	(*-----------------------Weiterschaltbedingungen----------------------------*)
	IF  NOT fb_xml_srv_read.bBusy  THEN
		IF NOT fb_xml_srv_read.bError THEN
			fb_state_entry.i16_next_step := 30;
		ELSE	(* Fehler *)
			s_PLC_Path_name:='!!! not found !!!';
			nErrId := fb_xml_srv_read.nErrId;
			fb_state_entry.i16_next_step := BEREIT;
			Error_:= TRUE;
		END_IF
	END_IF

	(*PLC Name und Pfad trennen *)
	s_PLC_name:=s_PLC_path_name;
	s_PLC_name:=s_PLC_path_name;
	len_str:=LEN(s_PLC_path_name);
	i:=0;

	FOR i:=1 TO len_str DO
		s_PLC_name:=DELETE(s_PLC_name,FIND(s_PLC_name,'\'),1);
	END_FOR

	s_PLC_path:=s_PLC_path_name;
	s_PLC_path:=DELETE(s_PLC_Path,LEN(s_PLC_path)-FIND(s_PLC_path,s_PLC_name)+1,FIND(s_PLC_path,s_PLC_name));
	s_Projekt_path:=s_PLC_path;

	len_str:=LEN(s_Projekt_path);
	s_Projekt_path:=LEFT(s_Projekt_path, len_str-1);

	(*PLC-Pfad löschen*)
	mid_str:='';
	len_str:=LEN(s_Projekt_path);
	FOR i:=1 TO LEN(s_Projekt_path) DO
			IF		mid_str <> '\' THEN
					s_Projekt_path:=LEFT(s_Projekt_path, len_str-i);
					mid_str:=MID(s_Projekt_path, 1 , len_str-i);
			END_IF
	END_FOR
(*=======================================================*)
30:  fb_state_entry.s_debugtext:='Pfade zusammen bauen';

	IF	s_Projekt_path <> '' THEN
		fb_state_entry.i16_next_step := BEREIT;
	END_IF

	IF	fb_state_entry.X THEN
		IF	FIND(s_tools_path,':') = 0 THEN
			s_tools_path:=CONCAT(s_Projekt_path,s_tools_path);
		END_IF

		IF	FIND(s_ud_path,':') = 0 THEN
			s_ud_path:=CONCAT(s_Projekt_path,s_ud_path);
		END_IF

		IF	FIND(MP_TDPathLocal,':') = 0 THEN
			MP_TDPathLocal:=CONCAT(s_Projekt_path,MP_TDPathLocal);
		END_IF

		IF	FIND(MP_TDPathService,':') = 0 THEN
			MP_TDPathService:=CONCAT(s_Projekt_path,MP_TDPathService);
		END_IF

		IF	FIND(MP_LocalDriveRoot,':') = 0 THEN
			MP_LocalDriveRoot:=CONCAT(s_Projekt_path,MP_LocalDriveRoot);
		END_IF

		IF	FIND(MP_ExportDrive,':') = 0 THEN
			MP_ExportDrive:=LEFT(s_PLC_path_name, 2);
		END_IF

		IF	FIND(MP_ExportDrivePathTD,'_') = 0 THEN
			MP_ExportDrivePathTD:=CONCAT(s_Projekt_path,MP_ExportDrivePathTD);
		END_IF

		IF	FIND(MP_ExportDrivePathMP,'_') = 0 THEN
			MP_ExportDrivePathMP:=CONCAT(s_Projekt_path,MP_ExportDrivePathMP);
		END_IF

		IF	FIND(LOG_RDPathLocal,':') = 0 THEN
			LOG_RDPathLocal:=CONCAT(s_Projekt_path,LOG_RDPathLocal);
		END_IF

		IF	FIND(LOG_ExportDrivePathRD,'_') = 0 THEN
			LOG_ExportDrivePathRD:=CONCAT(s_Projekt_path,LOG_ExportDrivePathRD);
		END_IF

	END_IF

(*=======================================================*)
BEREIT:  fb_state_entry.s_debugtext:='Warten auf Start';

	IF	fb_state_entry.E THEN
		Start:= FALSE;
		Done := TRUE;
	END_IF

	IF	Start THEN
		fb_state_entry.i16_next_step:=INIT;
	END_IF

	IF	fb_state_entry.X THEN
		Done := FALSE;
		Error_:= FALSE;
	END_IF

END_CASE

fb_state_entry(i16_pos:= 2);
(*========================================================================================*)

(* XML *)
fb_xml_srv_read(
	sNetId:= '',
	ePath:= PATH_GENERIC,
	nMode:= XMLSRV_SKIPMISSING,
	sSymName:= ,
	sFilePath:= ,
	sXPath:= ,
	bExecute:= ,
	tTimeout:= t#10s,
	bBusy=> ,
	bError=> ,
	nErrId=> );
END_PROGRAM

(* POU zLibrary/ept/min_exit/ST_MinExit, ST *)
PROGRAM ST_MinExit
VAR
	btn_min					: sButtonVisu;
	btn_exit					: sButtonVisu;

	fb_f_trig_minimieren		: F_TRIG;
	fb_tof_minimieren			: TOF;
	NT_StartProcess 			: NT_StartProcess;
	s_comndline						:STRING(255);
END_VAR
(*
in der C:\TwinCAT\Plc\TwinCAT PLC Control.ini muss
NoFullScreenMode=No umgestellt werden
=====================================================================*)



btn_min.Text:='_';
btn_min.Enable:=FALSE;
IF	btn_min.Pressed THEN
	btn_min.BackgroundColor:=Color.darkgrey;
ELSE
	btn_min.BackgroundColor:=Color.lightgrey;
END_IF
btn_min.TextColor:=Color.black;
btn_min.Visible:=FALSE;
fb_f_trig_minimieren(CLK:=btn_min.Pressed);
fb_tof_minimieren(IN:=fb_f_trig_minimieren.Q,PT:=t#1s);

IF	fb_f_trig_minimieren.Q THEN
	NT_StartProcess.START:=TRUE;
END_IF
IF 	NT_StartProcess.BUSY THEN
	NT_StartProcess.START:=FALSE;
END_IF

		(*minimieren wird mit vbs Skript gestartet*)
	NT_StartProcess(
			NETID:=,
			PATHSTR	:='C:\Windows\System32\wscript.exe',
			DIRNAME	:=s_tools_path,
			COMNDLINE	:='minimieren.vbs',
			START		:=,
			TMOUT		:=T#10s);
(*=====================================================================*)
btn_exit.Text:='X';
btn_exit.Enable:=FALSE;
IF	btn_exit.Pressed THEN
	btn_exit.BackgroundColor:=Color.darkgrey;
ELSE
	btn_exit.BackgroundColor:=Color.lightgrey;
END_IF

btn_exit.TextColor:=Color.black;
btn_exit.Visible:=FALSE;
END_PROGRAM

(* POU zLibrary/ept/ST_SaveAndLoad, ST *)
PROGRAM ST_SaveAndLoad
VAR_OUTPUT
	st_ctrl_out			:struct_ctrl_out;
END_VAR
VAR
	b_init				:BOOL;
	fb_state_entry		:ST_StateEntry;
	fb_ton_quitt		:TON;

	NT_StartProcess 	:NT_StartProcess;
	fbFileDelete		:FB_FileDelete;

	s_script			:STRING;

	btn_load			:sButtonVisu;
	btn_save			:sButtonVisu;

END_VAR
VAR CONSTANT
		s_bbgenMachineToSrv				:STRING:=		'_TD_save.bat';
		s_bbgenSrvToMachine				:STRING:=		'_TD_load.bat';

END_VAR
(*======================================================
   ST_SaveAndLoad
 ------------------------------------------------------
   Auth: 		Werner Friedl   						 
   Date: 		06.10.2020   						     
   Rev.: 		1.0	
   Desc:		Die bat Datein zum laden und speichern der BBgen Dateien werden hier ausgeführt.
			mit der Constante b_wkzBereinigen kann bestimmt werden, ob die Werkzeugdateu vorher gelöscht wird.

 ========================================================*)
IF	NOT b_init THEN
	b_Init:=TRUE;
END_IF
CallPrg();
Btn_init();
(* ========================================================*)
fb_ton_quitt(IN:= , PT:= t#100ms, Q=> , ET=> );

fb_state_entry(i16_pos:= 1);
CASE fb_state_entry.i16_step OF
(*=======================================================*)
INIT_OBJ:
		fb_state_entry.i16_next_step := INIT;

(*=======================================================*)
INIT:
	fb_state_entry.i16_next_step := BEREIT;

(*=======================================================*)
BEREIT:	fb_state_entry.s_debugtext:='warte auf Taster Save oder Load';

	IF fb_state_entry.E THEN
		st_ctrl_out.b_bereit:=TRUE;
		NT_StartProcess.START:=FALSE;
	END_IF

	(*-----------------------Weiterschaltbedingungen----------------------------*)
	IF 	btn_load.Pressed THEN
		fb_state_entry.i16_next_step:=110;
		s_script:=CONCAT(CURRENTLANGUAGE,s_bbgenSrvToMachine);
	ELSIF
		btn_save.Pressed THEN
		s_script:=CONCAT(CURRENTLANGUAGE,s_bbgenMachineToSrv);
		fb_state_entry.i16_next_step:=110;
	END_IF


	IF fb_state_entry.X THEN
		st_ctrl_out.b_busy:=TRUE;
		st_ctrl_out.b_bereit := FALSE;
		st_ctrl_out.b_fertig := FALSE;
	END_IF

(*=======================================================*)
110:fb_state_entry.s_debugtext:='start bat Script "Laden der Dateien vom Server"';

	IF 	fb_state_entry.E THEN
		NT_StartProcess.START:=TRUE;
	END_IF

	(*-----------------------Weiterschaltbedingungen----------------------------*)
	IF 	NT_StartProcess.BUSY THEN
		fb_state_entry.i16_next_step:=120;
	END_IF

	IF 	fb_state_entry.X THEN
		NT_StartProcess.START:=FALSE;
	END_IF

(*=======================================================*)
120:fb_state_entry.s_debugtext:='Warten auf fertig';

	IF	NOT btn_load.Pressed AND
		NOT btn_save.Pressed  THEN
		IF 	NT_StartProcess.ERR THEN
			fb_state_entry.s_debugtext:=CONCAT(fb_state_entry.s_debugtext,' ERRID => ');
			fb_state_entry.s_debugtext:=CONCAT(fb_state_entry.s_debugtext,UDINT_TO_STRING(NT_StartProcess.ERRID));
			fb_state_entry.i16_next_step:=FEHLER;
		ELSIF
			NOT NT_StartProcess.BUSY AND
			NOT NT_StartProcess.ERR AND
			fb_state_entry.fb_ton_Step.ET>t#3000ms THEN
			st_ctrl_out.b_busy:=FALSE;
			st_ctrl_out.b_fertig := TRUE;
			fb_state_entry.i16_next_step:=BEREIT;
		END_IF
	END_IF

(*=======================================================*)
STOP, FEHLER:

	IF fb_state_entry.E THEN
		st_ctrl_out.b_fehler := fb_state_entry.i16_step = FEHLER;
		st_ctrl_out.b_gestoppt := fb_state_entry.i16_step = STOP;
		st_ctrl_out.b_busy:=FALSE;
	END_IF

	IF	fb_state_entry.fb_ton_Step.ET > t#1000ms THEN   (*Quittiert sich selbst*)
		fb_state_entry.i16_next_step:=INIT;
	END_IF

END_CASE

fb_state_entry(i16_pos:= 2 );
END_PROGRAM
ACTION Btn_init:
btn_load.Text:='loadSrv';
btn_load.Enable:=CurrentUserLevel >=6 AND ModeSelect.Mode<=MODE_MANUAL;
IF btn_load.Enable THEN
	btn_load.TextColor:=Color.black;
ELSE
	btn_load.TextColor:=Color.grey;
END_IF
btn_load.Visible:= TRUE;

IF	btn_load.Pressed THEN
	btn_load.BackgroundColor:=Color.grey;
ELSE
	btn_load.BackgroundColor:=Color.lightgrey;
END_IF



btn_save.Text:='saveSrv';
btn_save.Enable:=CurrentUserLevel >=6 AND ModeSelect.Mode<=MODE_MANUAL;
IF btn_save.Enable THEN
	btn_save.TextColor:=Color.black;
ELSE
	btn_save.TextColor:=Color.grey;
END_IF
btn_save.Visible:= TRUE;

IF	btn_save.Pressed THEN
	btn_save.BackgroundColor:=Color.grey;
ELSE
	btn_save.BackgroundColor:=Color.lightgrey;
END_IF
END_ACTION
ACTION CallPrg:
NT_StartProcess(
	NETID:='',
	PATHSTR		:='C:\Windows\System32\cmd.exe',
	DIRNAME		:=s_tools_path,
	COMNDLINE	:=CONCAT('/C start /b ', s_script),
	START			:=,
	TMOUT			:=DEFAULT_ADS_TIMEOUT);


fbFileDelete(
	sNetId:= ,
	sPathName:= , 
	ePath:= PATH_GENERIC,
	bExecute:= ,
	tTimeout:= t#1s );
END_ACTION

(* POU zLibrary/ept/BDE/ST_Hydra8, ST *)
PROGRAM ST_Hydra8
VAR
	fb_tof_produktion			: TOF;
	fb_r_trig_signal			: R_TRIG;

	a_signal_produktion				AT %Q* : BOOL;
	a_signal_gutteil				AT %Q* : BOOL;
	a_signal_schlechtteil			AT %Q* : BOOL;
	a_signal_reserve				AT %Q* : BOOL;
	a_Fehlerfeld					: DWORD := 0;
END_VAR
(* Zeiten *)
fb_tof_produktion(
				IN:= 	(fb_r_trig_signal.Q AND
				ModeSelect.Mode=MODE_AUTO_RUN) OR
				(ST02_S1_40K01.BitInToCheck),
				PT:= T#60s,
				Q=>  a_signal_produktion,
				ET=> );

(* Flanken *)
IF	ST_CPU.LNG =CZ THEN
	fb_r_trig_signal(	CLK:= Robot01.State = STATE_OK);
END_IF

st_Hydra8Data.bStatus[_PRODUKTION] := a_signal_produktion;
END_PROGRAM

(* POU zLibrary/ept/BDE/ST_ImportHydraString, ST *)
PROGRAM ST_ImportHydraString
VAR_INPUT
	s_Path				: T_MaxString;
	sDateiName			: STRING;
	tStartTime			: TIME := T#10S;
END_VAR
VAR
	fb_state_entry			: ST_StateEntry;
	fbFindFiles			: FB_EnumFindFileList;
	fbFindFilesEntry		: ST_FindFileEntry;
	fbFileOpen			: FB_FileOpen;
	fbFileGets			: FB_FileGets;
	fbFileClose			: FB_FileClose;
	fbFileDelete			: FB_FileDelete;
	HelpString			: T_MaxString;
	fb_ton_start			: TON;
	hFile				:UINT:=0;
	nErrIdOpen			:UDINT;
	nErrIdRead			:UDINT;
	nErrIdClose			:UDINT;
	nErrIdDelete			:UDINT;
	sFileName			:STRING;

	iHelp				: INT;

	(* Für Anzeige in Visu *)
	iProduktionssperre	: INT;	(* 0 = nicht aktiv, 1 = aktiv, 2 = Status ungültig *)
END_VAR
VAR_OUTPUT
	Ready						:BOOL;
	Busy						:BOOL;
	Done						:BOOL;
	Error						:BOOL;
END_VAR
VAR CONSTANT
	sDatumPrefix				: STRING := 'DAT=';
	sZeitPrefix				: STRING := 'ZEI=';
	sOutput					: STRING := 'OUT';
	sTrennzeichen			: STRING := '|';
END_VAR
(*======================================================
   ST: ST_Import_Hydra_String
 ------------------------------------------------------
   Auth: 	Thomas Vilgis    						 
   Date: 	02.02.2022    						     
   Rev.: 	1.0	
   Desc:		Es wird alle 10 Sekunden (Zeit im Aufruf einstellbar) eine Textdatei mit 8 Status Ausgänge von Hydra erstellt.
			TwinCAT liest diese Datei aus und löscht sie dann.
			Es gibt nur eine Zeile in der Textdatei.
			Der erste Ausgang ist für den Status der Produktionssperre.
			Ein OUT Status steht nur in der Datei, wenn es eine Änderung gegeben hat.	
				
			So sieht die Datei aus: (alles in einer Zeile)
			OUT1=0|OUT2=0|OUT3=0|OUT4=0|OUT5=0|
			OUT6=0|OUT7=0|OUT8=0|DAT=02.02.2021|ZEI=07:16:00

   Historie: 	1.0

 ========================================================*)



(* Zeiten *)
fb_ton_start(IN:= NOT fb_ton_start.Q, PT:= tStartTime, Q=>  , ET=> );


(* ======================================Schrittkette======================================== *)
fb_state_entry(i16_pos:= 1);

CASE fb_state_entry.i16_step OF
(*=======================================================*)
	INIT_OBJ: fb_state_entry.s_debugtext:='initialisieren';

		(*-----------------------Weiterschaltbedingungen----------------------------*)
		IF fb_state_entry.fb_ton_Step.ET >= T#5S THEN
			fb_state_entry.i16_next_step:=BEREIT;
		END_IF

(*=======================================================*)
	BEREIT: fb_state_entry.s_debugtext:='Start';

		IF fb_state_entry.E THEN
			Ready := TRUE;
		END_IF

		(*-----------------------Weiterschaltbedingungen----------------------------*)
		IF fb_ton_start.Q THEN
			Error := FALSE;
			Busy := TRUE;
			Ready := FALSE;
			Done := FALSE;
			fb_state_entry.i16_next_step:=110;
		END_IF
		
		IF fb_state_entry.X THEN
			sFileName:=CONCAT(s_Path,sDateiName);
		END_IF
		
(*=======================================================*)
	110: fb_state_entry.s_debugtext:='HelpString löschen';
	
		IF fb_state_entry.E THEN
			HelpString := '';
		END_IF

		(*-----------------------Weiterschaltbedingungen----------------------------*)
		fb_state_entry.i16_next_step:=120;

(*=======================================================*)
	120: fb_state_entry.s_debugtext:='Prüfe, ob Datei vorhanden ist';

		IF fb_state_entry.E THEN
			fbFindFiles.bExecute := TRUE;
		END_IF

		(*-----------------------Weiterschaltbedingungen----------------------------*)
		IF fbFindFiles.bBusy THEN
			fb_state_entry.i16_next_step:=130;
		END_IF

(*=======================================================*)
	130: fb_state_entry.s_debugtext:='Prüfe, ob Datei vorhanden ist';

		(*-----------------------Weiterschaltbedingungen----------------------------*)
		IF NOT fbFindFiles.bBusy THEN
			fbFindFiles.bExecute := FALSE;
			IF NOT fbFindFiles.bError THEN
				IF fbFindFiles.nFindFiles = 1 THEN
					fb_state_entry.i16_next_step:=140;
				ELSE
					fb_state_entry.i16_next_step:=240;	(* Datei nicht vorhanden >> Auswertung *)
				END_IF
			ELSE
				fb_state_entry.i16_next_step:=FEHLER;
			END_IF
		END_IF

(*=======================================================*)
	140: fb_state_entry.s_debugtext:='Datei öffnen';

		IF fb_state_entry.E THEN
		   	fbFileOpen.bExecute:=TRUE;
		END_IF

		(*-----------------------Weiterschaltbedingungen----------------------------*)
		IF fbFileOpen.bBusy THEN
			fb_state_entry.i16_next_step:=150;
		END_IF

(*=======================================================*)
	150: fb_state_entry.s_debugtext:='Datei öffnen';

		(*-----------------------Weiterschaltbedingungen----------------------------*)
		IF 	NOT fbFileOpen.bBusy THEN

			fbFileOpen.bExecute:=FALSE;
			IF 	fbFileOpen.bError THEN
				nErrIdOpen:=fbFileOpen.nErrId;
				fb_state_entry.i16_next_step:=200;
			ELSE
				hFile := fbFileOpen.hFile;	(* Sehr wichtig hFile für FileRead und Fileclose übergeben *)
				fb_state_entry.i16_next_step:=160;
			END_IF
		END_IF

(*=======================================================*)
	160: fb_state_entry.s_debugtext:='Datei auslesen';

		IF fb_state_entry.E THEN
			fbFileGets.bExecute:=TRUE;
		END_IF

		(*-----------------------Weiterschaltbedingungen----------------------------*)
		IF  fbFileGets.bBusy THEN
			fb_state_entry.i16_next_step:=170;
		END_IF

(*=======================================================*)
	170: fb_state_entry.s_debugtext:='Datei auslesen';

		(*-----------------------Weiterschaltbedingungen----------------------------*)
		IF 	NOT fbFileGets.bBusy THEN
			fbFileGets.bExecute:=FALSE;
			IF 	fbFileGets.bError THEN
				nErrIdRead:=fbFileGets.nErrId;
				fb_state_entry.i16_next_step:=200;
			ELSE
				HelpString := fbFileGets.sLine;
				fb_state_entry.i16_next_step:=200;
			END_IF
		END_IF

(*=======================================================*)
	200: fb_state_entry.s_debugtext:='Datei schließen';

		IF fb_state_entry.E THEN
			fbFileClose.bExecute:=TRUE;
		END_IF

		(*-----------------------Weiterschaltbedingungen----------------------------*)
		IF 	fbFileClose.bBusy THEN
			fb_state_entry.i16_next_step:=210;
		END_IF

(*=======================================================*)
	210: fb_state_entry.s_debugtext:='Datei schließen';

		(*-----------------------Weiterschaltbedingungen----------------------------*)
		IF NOT fbFileClose.bBusy THEN
			fbFileClose.bExecute:=FALSE;
			IF 	fbFileClose.bError THEN
				nErrIdClose:=fbFileClose.nErrId;
				fb_state_entry.i16_next_step:=FEHLER;
			ELSE
				hFile := 0;
				fb_state_entry.i16_next_step:=220;
			END_IF
		END_IF
		
(*=======================================================*)
	220: fb_state_entry.s_debugtext:='Datei löschen';

		IF fb_state_entry.E THEN
			fbFileDelete.bExecute:=TRUE;
		END_IF

		(*-----------------------Weiterschaltbedingungen----------------------------*)
		IF 	fbFileDelete.bBusy THEN
			fb_state_entry.i16_next_step:=230;
		END_IF

(*=======================================================*)
	230: fb_state_entry.s_debugtext:='Datei löschen';

		(*-----------------------Weiterschaltbedingungen----------------------------*)
		IF NOT fbFileDelete.bBusy THEN
			fbFileDelete.bExecute:=FALSE;
			IF 	fbFileDelete.bError THEN
				nErrIdDelete:=fbFileDelete.nErrId;
				fb_state_entry.i16_next_step:=FEHLER;
			ELSE
				fb_state_entry.i16_next_step:=240;
			END_IF
		END_IF

(* Falls die Auswertung der Datei für jede Anlage unterschiedlich ist,
sollte man die Auswertung in einem eigenen Baustein machen *)
(*=======================================================*)
	240: fb_state_entry.s_debugtext:='Auswertung, ob Produktionssperre aktiv ist';

		IF fb_state_entry.E THEN
			IF fbFindFiles.nFindFiles = 0 THEN	(* Datei war gar nicht vorhanden *)
				iProduktionssperre := 2;	(* Status ungültig *)
			ELSE
				(* Suche nach OUT1= *)
				iHelp := FIND(HelpString, CONCAT(sOutput, '1='));
				IF iHelp > 0 THEN
					IF MID(HelpString, 1, 6) = '0' THEN	(* an Stelle 6 steht 0 oder 1 *)
						iProduktionssperre := 0;	(* nicht aktiv *)
					ELSIF MID(HelpString, 1, 6) = '1' THEN	(* an Stelle 6 steht 0 oder 1 *)
						iProduktionssperre := 1;	(* aktiv *)
					END_IF
				END_IF
			END_IF
		END_IF

		(*-----------------------Weiterschaltbedingungen----------------------------*)
		Busy := FALSE;
		Done := TRUE;
		fb_state_entry.i16_next_step:=BEREIT;
		
	

(*=======================================================*)
	FEHLER:
		IF fb_state_entry.E THEN
			Error := TRUE;
		END_IF

		(*-----------------------Weiterschaltbedingungen----------------------------*)
		fb_state_entry.i16_next_step:=BEREIT;

END_CASE


fb_state_entry(i16_pos:= 2);


fbFindFiles(
	bExecute	:= ,
	sNetId		:= '',
	sPathName	:= sFileName,
	pFindList	:= ADR(fbFindFilesEntry),
	cbFindList	:= SIZEOF(fbFindFilesEntry),
	tTimeout	:= t#1s );

 fbFileOpen(
	sNetId:='',
	sPathName:= sFileName,
	nMode:=FOPEN_MODEREAD,
	ePath:=PATH_GENERIC,
	bExecute:= ,
	tTimeout:=T#1s,
	hFile=> );

fbFileGets(
	sNetId:= , 
	hFile:= hFile, 
	bExecute:= , 
	tTimeout:= , 
	bBusy=> , 
	bError=> , 
	nErrId=> , 
	sLine=> , 
	bEOF=> );

fbFileClose(
	sNetId:='',
	hFile:=hFile,
	bExecute:= ,
	tTimeout:=T#1S);
	
fbFileDelete(
	sNetId:= , 
	sPathName:= sFileName, 
	ePath:= PATH_GENERIC, 
	bExecute:= , 
	tTimeout:= , 
	bBusy=> , 
	bError=> , 
	nErrId=> );
END_PROGRAM

(* POU System/LoginDialog/ImpExp_UD, ST *)
PROGRAM ImpExp_UD
VAR_INPUT
	Start_write				:BOOL;
	Start_read				:BOOL;
	path					:STRING(255);
	filename					:STRING(255);
END_VAR
VAR
	b_init					:BOOL;
	fb_state_entry				:ST_StateEntry;

	fb_xml_srv_read			: FB_XmlSrvReadByName;
	fb_xml_srv_write			: FB_XmlSrvWriteByName;

	fb_rtrig_Start_read			:R_TRIG;
	fb_rtrig_Start_write_to_server:R_TRIG;
	fb_ton_init				:TON;
	fb_ton_wz				:TON;
	fb_ton_uez				:TON;

	bError					: BOOL;
	nErrId					: UDINT;
	s_info					: STRING;
	MsgOK					: BOOL;
	MsgID					:STRING(20);

	UserList_Copy			: ARRAY [1..NO_OF_USERS] OF sUserData;

END_VAR

VAR_OUTPUT
	Busy					:BOOL;
	Done					:BOOL;
	Error					:BOOL;
	ErrorMsg				:STRING(255);
END_VAR

VAR CONSTANT
	SymName				:STRING:='.UD';
	xPath					:STRING:='/UD';
END_VAR

VAR_IN_OUT

END_VAR
(*======================================================
   PRG: XML Import und Export der UD
 ------------------------------------------------------
   Auth: 		Werner Friedl    						 
   Date: 		05.01.2021  						     
   Rev.: 		1.0	
   Desc:		
	- Userdate werden beim Neustart eingelesen
	- bei einer Änderung wird Änderung automatisch in die xml eingeragen

   Historie:   1.0

 ========================================================*)
fb_ton_init(IN:= TRUE, PT:=t#1500ms , Q=> , ET=> );
IF	NOT b_init AND fb_ton_init.Q THEN
	Start_read := TRUE;
	b_Init:=TRUE;
END_IF

(* ========================================================*)
fb_rtrig_Start_read();
IF	fb_rtrig_Start_read.Q AND
	NOT Start_write THEN
	Start_read:=TRUE;
END_IF

IF 	(MEMCMP(ADR(UserList_Copy),ADR(UD.UserList),SIZEOF(UserList_Copy))<>0)AND (*automatisch speichern im Manualmode*)
     	ModeSelect.Mode <=MODE_MANUAL AND
	NOT Start_read AND
	b_Init THEN
	Start_write := TRUE;
END_IF

(* ========================================================*)
fb_ton_wz(IN:= , PT:=t#3000ms , Q=> , ET=> );
IF	fb_ton_wz.Q THEN
	fb_ton_wz.IN:=FALSE;
	s_info := '';
END_IF

fb_state_entry(i16_pos:= 1);
CASE fb_state_entry.i16_step OF

(*=======================================================*)
0:	(*initialisieren*)
	Start_write := FALSE;
	Start_read := FALSE;
	fb_state_entry.i16_next_step:=BEREIT;

(*=======================================================*)
BEREIT: fb_state_entry.s_debugtext:='warte auf start';

	IF	Start_read THEN
		fb_state_entry.i16_next_step:=110;
	END_IF

	IF	Start_write THEN
		fb_state_entry.i16_next_step:=200;
	END_IF

	IF fb_state_entry.X THEN
		fb_ton_uez.IN:=FALSE;
		Start_write:=FALSE;
		Start_read:=FALSE;
		Busy:=TRUE;
		Error:=FALSE;
		Done:=FALSE;
		nErrId:=0;
		ErrorMsg:='';
		MsgID:='';
	END_IF

(*=======================================================*)
110: fb_state_entry.s_debugtext:='XML auslesen';	 

	IF fb_state_entry.E THEN
		fb_xml_srv_read.sFilePath := CONCAT(path,filename);
		fb_xml_srv_read.sSymName:=SymName;
		fb_xml_srv_read.sXPath :=xPath;
		fb_xml_srv_read.bExecute := TRUE;
	END_IF

	IF fb_xml_srv_read.bBusy THEN
		fb_xml_srv_read.bExecute := FALSE;
		fb_state_entry.i16_next_step := 120;
	END_IF

(*=======================================================*)
120: fb_state_entry.s_debugtext:='Lesevorgang erfolgreich?';

	IF  NOT fb_xml_srv_read.bBusy  THEN
		IF NOT fb_xml_srv_read.bError THEN
			fb_state_entry.i16_next_step := 900;
		ELSE	(* Fehler *)
			nErrId := fb_xml_srv_read.nErrId;
			IF	nErrId =1804 THEN
				MsgID:='PM15';
				ErrorMsg:='Die Datei UD.xml ist nicht vorhanden';
				fb_state_entry.i16_next_step := 200;	(*Datei wird erstellt*)
			ELSE
				MsgID:='PM16';
				ErrorMsg:='Fehler beim Einlesen der UD.xml Datei';
				fb_state_entry.i16_next_step := FEHLER;
			END_IF
		END_IF
	END_IF

	IF fb_state_entry.X THEN
		fb_ton_wz.IN:=TRUE;
		s_info:=CONCAT('read ',filename);
	END_IF

(*=======================================================*)
200: fb_state_entry.s_debugtext:='XML schreiben';

	IF fb_state_entry.E THEN
		fb_xml_srv_write.sFilePath := CONCAT(path,filename);
		fb_xml_srv_write.sSymName:=SymName;
		fb_xml_srv_write.sXPath :=xPath;
		fb_xml_srv_write.bExecute := TRUE;
	END_IF

	IF fb_xml_srv_write.bBusy THEN
		fb_xml_srv_write.bExecute := FALSE;
		fb_state_entry.i16_next_step := 220;
	END_IF

(*=======================================================*)
220: fb_state_entry.s_debugtext:='Schreiben erfolgreich?';

	IF  NOT fb_xml_srv_write.bBusy  THEN
		IF NOT fb_xml_srv_write.bError THEN
			UserList_Copy := UD.UserList;
			fb_state_entry.i16_next_step := 900;
		ELSE	(* Fehler *)
			nErrId := fb_xml_srv_write.nErrId;
			MsgID:='PM17';
			ErrorMsg:='Fehler beim Schreiben der UD.xml';
			fb_state_entry.i16_next_step := FEHLER;
		END_IF
	END_IF

	IF fb_state_entry.X THEN
		fb_ton_wz.IN:=TRUE;
		fb_ton_uez.IN:=TRUE;		(*automatisch auf Server speichern*)
		s_info:=CONCAT('write ',filename);
	END_IF

(*=======================================================*)
900: fb_state_entry.s_debugtext:='Fertig';

	Busy:=FALSE;
	Done:=TRUE;
	fb_state_entry.i16_next_step:=0;

(*=======================================================*)
FEHLER:

	IF fb_state_entry.E THEN
		MessageHandler.ClearMessageLines(sVisu:=Visu.Message);
	END_IF
	MessageHandler.Msg.ID:=MsgID;
	MessageHandler.Msg.Name:=ErrorMsg;
	MessageHandler.Msg.Text:=ErrorMsg;
	MessageHandler.Msg.Color:=Color.red;
	MessageHandler.Msg.Station:=0;

	MessageHandler(
		Prio:=2, 							(*1=highest, .. , 4=lowest*)
		Btn1Addr:=ADR(MsgOk),			(*Address of Button1 , if Zero then Button is unvisible*)
		Btn2Addr:=,						(*Address of Button2 , if Zero then Button is unvisible*)
		sVisu:=Visu.Message);

	IF MsgOK THEN
		MsgOk:=FALSE;
		fb_state_entry.i16_next_step:=0;
		Busy:=FALSE;
		Error:=TRUE;
	END_IF
END_CASE

fb_state_entry(i16_pos:= 2);


fb_xml_srv_read(
	sNetId:= '',
	ePath:= PATH_GENERIC,
	nMode:= XMLSRV_SKIPMISSING,
	sSymName:= ,
	sFilePath:= ,
	sXPath:= ,
	bExecute:= ,
	tTimeout:= t#10s,
	bBusy=> ,
	bError=> ,
	nErrId=> );

fb_xml_srv_write(
	sNetId:= '',
	ePath:= PATH_GENERIC,
	nMode:= XMLSRV_ADDMISSING,
	sSymName:=  ,
	sFilePath:= ,
	sXPath:= ,
	bExecute:= ,
	tTimeout:= t#10s,
	bBusy=> ,
	bError=> ,
	nErrId=> );


(*automatisch auf Server speichern=============================================*)
fb_ton_uez(PT:=t#20s);
fb_rtrig_Start_write_to_server(CLK:=fb_ton_uez.Q , Q=> );
(*
NT_StartProcess(
	NETID:='',
	PATHSTR	:='C:\Windows\System32\cmd.exe',
	DIRNAME	:='D:\Tools ',
	COMNDLINE	:='/C copy C:\MP\MachPara.xml \\10.16.50.9\bbgen\UML3\MD & @ping localhost -n 4 >NUL',
	START		:=fb_rtrig_Start_write_to_server.Q,
	TMOUT		:=t#10s);
*)
(*
NT_StartProcess(
	NETID:='',
	PATHSTR	:='C:\Windows\System32\wscript.exe',
	DIRNAME	:='D:\Tools',
	COMNDLINE	:='de_PD_aktuell_von_uml_nach_server.vbs',
	START		:=fb_rtrig_Start_write_to_server.Q,
	TMOUT		:=t#10s);
*)
END_PROGRAM

(* POU System/LoginDialog/UserLoginHandler, ST *)
PROGRAM UserLoginHandler
VAR
	Keypad								: UserLoginKeypad;
	btn_Login							: VisuButton;
	btn_LogOut							: VisuButton;
	btn_ChangeUserData				: VisuButton;
	btn_ChangePassword				: VisuButton;

	PasswordChangeActive				: BOOL;

	UserListIndexFixed					: INT;
	FixUserList							: BOOL;
	FP_FixUserList						: R_TRIG;
	FP_PasswordChangeActive			: R_TRIG;

	SelectedUser						: sUserData;
	UserLoggedOut						: sUserData;
	EmptyUser							: sUserData;

	CurrentVisuOld						: STRING;
	UserListIndexOld					: INT;

	InfoLogin              					: ErrorStruct;
	InfoLogout           					: ErrorStruct;

	TP_LogegdIn						: TP;
	TP_LogegdOut						: TP;

	Index								: INT;

	ton_AutoLoggedOut					: TON;
	b_Button							: BOOL;
	CopyCurrentVisu						: STRING;
	s_AutoLoggedOut					: STRING;

END_VAR
VAR_IN_OUT
	sVisu								: sVisuLoginDialog;
	UserList								: ARRAY [1..NO_OF_USERS] OF sUserData;

END_VAR
VAR_OUTPUT
	CurrentUser							: sUserData;
	UserLoggedIn						: BOOL;
END_VAR
(* Fix Administrator and Operator *)
UserList[1].UserName							:= 'Administrator';
(*UserList[1].UserPassword						:= '123';*)			(*PW in der ".....\UD\UserList.xml  " ändern und PLC neu starten*)
UserList[1].UserLevel							:= 7;
UserList[1].UserCanChangeOwnPassword			:= FALSE;

UserList[2].UserName							:= 'Service';
UserList[2].UserLevel							:= 6;
UserList[2].UserCanChangeOwnPassword			:= FALSE;

(* Fix UserLoggedOut *)
UserLoggedOut.UserName						:= 'Produktion';(*'Logged out';*)
UserLoggedOut.UserPassword					:= '';
UserLoggedOut.UserLevel						:= 1;
UserLoggedOut.UserCanChangeOwnPassword	:= FALSE;



Keypad(sVisu:= sVisu.LoginKeyPad,HidePasswordString:=NOT PasswordChangeActive);

FixUserList:= Keypad.Visible OR
			(CurrentUser.UserName<>UserLoggedOut.UserName AND CurrentUserLevel<6);

FP_FixUserList(CLK:= FixUserList );


(* Save Selecte UserIndex from Visu *)
IF 	FP_FixUserList.Q THEN
	UserListIndexFixed:=sVisu.UserListIndex;
END_IF;

(* Disable Selection in sVisu  *)
IF 	FixUserList THEN
	sVisu.UserListIndex:=UserListIndexFixed;
ELSE
	IF	sVisu.UserListIndex > 0 THEN
		SelectedUser:=UserList[sVisu.UserListIndex];
	END_IF
END_IF


(* Handle Keypad *)
FP_PasswordChangeActive(CLK:= PasswordChangeActive);
IF 	btn_Login.PressedFlag AND SelectedUser.UserPassword<>'' OR	(*Login with PW*)
	FP_PasswordChangeActive.Q THEN								(*PW-Change*)
	Keypad.Visible:=TRUE;
END_IF

IF 	Keypad.btnESC OR Keypad.btnOK OR CurrentVisuOld<>CurrentVisu THEN
	Keypad.Visible:=FALSE;
END_IF


(* Handle Login / Logout *)
btn_Login	(TextOn:= 'Login',	Button:= sVisu.btn_Login );
btn_LogOut	(TextOn:= 'Logout',	Button:= sVisu.btn_LogOut );

btn_Login.Enable:=TRUE;

btn_LogOut.Enable:=CurrentUser.UserName<>UserLoggedOut.UserName AND NOT PasswordChangeActive;


IF btn_LogOut.PressedFlag THEN
	(* Generate information Errorlog *)
	InfoLogout.Text			:=  CONCAT('LoginHandler: User ausgeloggt:',CurrentUser.UserName);
	InfoLogout.Typ			:=  2;
	InfoLogout.No			:=  1;
	InfoLogout.DateTime	:=  gVarDTSystemtime;
	TP_LogegdOut.IN		:= TRUE;

	CurrentUserLevel		:= 0;
	CurrentUser				:= UserLoggedOut;
END_IF

(*LogIn finished ok*)
IF 	Keypad.btnOK AND Keypad.InputString=SelectedUser.UserPassword AND NOT PasswordChangeActive OR		(*Login with PW, and PW ok*)
	btn_Login.PressedFlag AND SelectedUser.UserPassword='' THEN												(*Login without PW*)
	CurrentUserLevel		:= SelectedUser.UserLevel;
	CurrentUser				:= SelectedUser;
	(* Generate information Errorlog *)
	InfoLogin.Text			:= CONCAT('LoginHandler: User eingeloggt:',CurrentUser.UserName);
	InfoLogin.Typ			:= 2;
	InfoLogin.No			:= 1;
	InfoLogin.DateTime		:= gVarDTSystemtime;
	TP_LogegdIn.IN			:= TRUE;
END_IF


(* Edit Userlist *)

(* Show Edit Fields *)
sVisu.ShowEditFields:=(sVisu.UserListIndex>=2 AND CurrentUserLevel=7) OR (sVisu.UserListIndex>=3 AND CurrentUserLevel=6);

btn_ChangeUserData(Button:= sVisu.btn_ChangeUserData );
btn_ChangeUserData.Visible:=sVisu.ShowEditFields;

IF 	sVisu.UserEdit.UserName='' THEN
	btn_ChangeUserData.TextOn:= 'ChangeUserDataDel';
ELSE
	btn_ChangeUserData.TextOn:= 'ChangeUserData';
END_IF

IF 	btn_ChangeUserData.PressedFlag THEN
	(* Take new Userdatas when Username is not Administrator and Produktion *)
	IF 	sVisu.UserEdit.UserName <> 'Administrator' AND sVisu.UserEdit.UserName <> 'Produktion' THEN
		UserList[sVisu.UserListIndex]:=sVisu.UserEdit;
		IF 	UserList[sVisu.UserListIndex].UserName=''  THEN
			FOR index:= sVisu.UserListIndex TO DINT_TO_INT(NO_OF_USERS-1) BY 1 DO
				UserList[index]:=UserList[index+1];
			END_FOR
				UserList[index]:=EmptyUser;
		END_IF
	END_IF
END_IF

IF UserListIndexOld<>sVisu.UserListIndex
THEN
sVisu.UserEdit:=UserList[sVisu.UserListIndex];
END_IF

(* Change own Password from Allowed User *)
btn_ChangePassword(TextOn:= 'Passwortändern',Button:= sVisu.btn_ChangePassword );
btn_ChangePassword.Visible:=CurrentUser.UserCanChangeOwnPassword AND CurrentUser.UserName=SelectedUser.UserName;

IF 	btn_ChangePassword.PressedFlag THEN
	PasswordChangeActive:=TRUE;
END_IF

IF 	PasswordChangeActive	AND
	(Keypad.btnESC OR Keypad.btnOK OR CurrentVisuOld<>CurrentVisu) THEN
	IF Keypad.btnOK THEN
		UserList[sVisu.UserListIndex].UserPassword:=Keypad.InputString;
	END_IF
	PasswordChangeActive:=FALSE;
	Keypad.Visible:=FALSE;
END_IF

(* Compare Userleve with CurrentUser *)
IF 	CurrentUserLevel <> CurrentUser.UserLevel THEN
	CurrentUserLevel := CurrentUser.UserLevel;
END_IF

(* Check Current Username not Empty *)
IF  	CurrentUser.UserName = '' THEN
	CurrentUser := UserLoggedOut;
END_IF


UserLoggedIn:= (CurrentUser.UserName <> UserLoggedOut.UserName);


(* Last Operation!!!! *)
UserListIndexOld:=sVisu.UserListIndex;
CurrentVisuOld:=CurrentVisu;

IF 	TP_LogegdIn.Q THEN
	ErrorHandler.AddError(ErrorToAdd:=InfoLogin,sVisu:=Visu.ErrorHandler);
END_IF

IF 	TP_LogegdOut.Q THEN
	ErrorHandler.AddError(ErrorToAdd:=InfoLogout,sVisu:=Visu.ErrorHandler);
END_IF

TP_LogegdIn(PT:= t#1s );
TP_LogegdOut(PT:= t#1s );

TP_LogegdIn.IN:=FALSE;
TP_LogegdOut.IN:=FALSE;

(*========Benutzer automatisch abmelden=================================*)

b_Button:=
	Visu.ModeSelect.BtnManual.Pressed OR
	Visu.ModeSelect.BtnAuto.Pressed OR
	Visu.ModeSelect.BtnAutoStart.Pressed OR
	Visu.ModeSelect.BtnAutoStop.Pressed OR
	Visu.ModeSelect.BtnSpecial.Pressed OR
	Visu.ModeSelect.BtnRunEmpty.Pressed OR
	Visu.ModeSelect.BtnStepCycle.Pressed OR
	Visu.ModeSelect.BtnSpecial.Pressed OR
	Visu.ModeSelect.BtnSpecStep.Pressed OR
	Visu.ModeSelect.BtnHomeRun.Pressed OR
	Visu.ModeSelect.BtnReset.Pressed;

IF	CurrentVisu<>CopyCurrentVisu THEN
	b_Button:=TRUE;
	CopyCurrentVisu:=CurrentVisu;
END_IF

IF	CurrentUser.UserName<>UserLoggedOut.UserName AND
	MP.ST00.MaxLogInTime <> 0 THEN

	ton_AutoLoggedOut(
			IN:=NOT  b_Button,
			PT:=DINT_TO_TIME(MP.ST00.MaxLogInTime*60000) ,
			Q=> ,
			ET=> );
	s_AutoLoggedOut:=ET_TO_STRING(ton_AutoLoggedOut.PT - ton_AutoLoggedOut.ET);
	s_AutoLoggedOut:=LEFT(s_AutoLoggedOut,FIND( s_AutoLoggedOut,'s'));

	IF	ton_AutoLoggedOut.Q THEN
		(* Generate information Errorlog *)
		InfoLogout.Text                 := CONCAT('LoginHandler: User ausgeloggt:',CurrentUser.UserName);
		InfoLogout.Typ                  := 2;
		InfoLogout.No                   := 1;
		InfoLogout.DateTime         := gVarDTSystemtime;
		TP_LogegdOut.IN:=TRUE;

		CurrentUserLevel		:=1;
		CurrentUser				:=UserLoggedOut;
	END_IF

ELSE
	ton_AutoLoggedOut(IN:=FALSE);
	s_AutoLoggedOut:='';
END_IF
END_PROGRAM

(* POU System/LoginDialog/UserLoginKeypad, ST *)
FUNCTION_BLOCK UserLoginKeypad
VAR
	btn_Key1					: VisuButton;
	btn_Key2					: VisuButton;
	btn_Key3					: VisuButton;
	btn_Key4					: VisuButton;
	btn_Key5					: VisuButton;
	btn_Key6					: VisuButton;
	btn_Key7					: VisuButton;
	btn_Key8					: VisuButton;
	btn_Key9					: VisuButton;
	btn_Key0					: VisuButton;
	btn_KeyDot				: VisuButton;

	btn_KeyBack				: VisuButton;
	btn_KeyEsc				: VisuButton;
	btn_KeyClear			: VisuButton;
	btn_KeyOK					: VisuButton;
	btn_KeyVorzeichen	: VisuButton;

	InputStringLen		: INT;
	I									: INT;

	FP_Init						:	R_TRIG;
END_VAR
VAR_IN_OUT
	sVisu							: sNumericKeypad;
END_VAR
VAR_INPUT
	Visible						:	BOOL;
	HidePasswordString: BOOL;
END_VAR
VAR_OUTPUT
	InputString				:	STRING;
	btnOK							:	BOOL;
	btnESC						:	BOOL;
END_VAR
btn_Key0(	TextOn:= '0',	Button:= sVisu.btn_Key0 );
btn_Key1(	TextOn:= '1',	Button:= sVisu.btn_Key1 );
btn_Key2(	TextOn:= '2',	Button:= sVisu.btn_Key2 );
btn_Key3(	TextOn:= '3',	Button:= sVisu.btn_Key3 );
btn_Key4(	TextOn:= '4',	Button:= sVisu.btn_Key4 );
btn_Key5(	TextOn:= '5',	Button:= sVisu.btn_Key5 );
btn_Key6(	TextOn:= '6',	Button:= sVisu.btn_Key6 );
btn_Key7(	TextOn:= '7',	Button:= sVisu.btn_Key7 );
btn_Key8(	TextOn:= '8',	Button:= sVisu.btn_Key8 );
btn_Key9(	TextOn:= '9',	Button:= sVisu.btn_Key9 );
btn_KeyBack(	TextOn:= 'Back',	Button:= sVisu.btn_KeyBack );
btn_KeyEsc(	TextOn:= 'Esc',	Button:= sVisu.btn_KeyEsc );
btn_KeyClear(	TextOn:= 'Clear',	Button:= sVisu.btn_KeyClear );
btn_KeyOK(	TextOn:= 'OK',	Button:= sVisu.btn_KeyOK );

btn_KeyDot(	TextOn:= '.',	Button:= sVisu.btn_KeyDot );
btn_KeyVorzeichen(	TextOn:= '+/-',	Button:= sVisu.btn_KeyVorzeichen );

btn_KeyDot.Enable:=FALSE;
btn_KeyVorzeichen.Enable:=FALSE;

svisu.Visible:=Visible;
svisu.Enable:=Visible;

(* initialize  *)
FP_Init(CLK:= Visible);

IF FP_Init.Q
THEN
	InputString:='';
END_IF


InputStringLen:=LEN(InputString);

IF btn_Key0.PressedFlag
THEN
	InputString:=CONCAT(InputString,'0');
END_IF
IF btn_Key1.PressedFlag
THEN
	InputString:=CONCAT(InputString,'1');
END_IF
IF btn_Key2.PressedFlag
THEN
	InputString:=CONCAT(InputString,'2');
END_IF
IF btn_Key3.PressedFlag
THEN
	InputString:=CONCAT(InputString,'3');
END_IF
IF btn_Key4.PressedFlag
THEN
	InputString:=CONCAT(InputString,'4');
END_IF
IF btn_Key5.PressedFlag
THEN
	InputString:=CONCAT(InputString,'5');
END_IF
IF btn_Key6.PressedFlag
THEN
	InputString:=CONCAT(InputString,'6');
END_IF
IF btn_Key7.PressedFlag
THEN
	InputString:=CONCAT(InputString,'7');
END_IF
IF btn_Key8.PressedFlag
THEN
	InputString:=CONCAT(InputString,'8');
END_IF
IF btn_Key9.PressedFlag
THEN
	InputString:=CONCAT(InputString,'9');
END_IF

IF btn_KeyBack.PressedFlag
THEN
	InputString:=LEFT(InputString,InputStringLen-1);
END_IF

IF btn_KeyClear.PressedFlag
THEN
	InputString:='';
END_IF

IF btn_KeyEsc.PressedFlag
THEN
	InputString:='';
END_IF

InputStringLen:=LEN(InputString);
svisu.InputString:='';

IF HidePasswordString
THEN

	FOR i:=1 TO InputStringLen DO
		svisu.InputString:=CONCAT(svisu.InputString,'*');
	END_FOR
ELSE
	svisu.InputString:=InputString;
END_IF
btnOK:=btn_KeyOK.PressedFlag;
btnESC:=btn_KeyEsc.PressedFlag;
END_FUNCTION_BLOCK

(* POU System/TDHandler/TDHandler, ST *)
PROGRAM TDHandler
VAR

	WriteXML					: FB_XmlSrvWriteByName;
	ReadXML					: FB_XmlSrvReadByName;
	DeleteXML					: FB_FileDelete;
	DeleteXMLactive			: BOOL;

	FindFiles					: FB_EnumFindFileList;

	filesList						: ARRAY[1..NO_OF_FILES] OF ST_FindFileEntry;

	i,j							: DINT;

	FileNameWrite				: STRING(255);
	FileNameRead				: STRING(255);
	FileNameDelete				: STRING(255);

	FileWriteSource				: STRING(255);
	FileReadTarget				: STRING(255);


	FileNameSearch				: STRING(255);

	FileFilterOld					: STRING(255);
	FileIndexOld					: DINT;
	fb_rTrigFilList				: R_TRIG;

	BtnSaveAs					: VisuButton;
	BtnActivate					: VisuButton;
	BtnDelete					: VisuButton;

	FirstCycle					: BOOL;
	SetActivate					: BOOL := FALSE;

	Error						: ErrorStruct;
	ErrorElapsed				: R_TRIG;
	TDValid						: BOOL;
	FileNameReadCopy			: STRING(255);
	TDCopy						: sTypeData;
	TDempty					: sTypeData;
	TypeNameCopy				: STRING;
	fb_ExpActTDNo				: FB_ExporString;	(* Fehlermeldungen in Errorlog (txt) schreiben *)

	b_Dialog_save_as_on		: BOOL;

	s_Xpath						: T_MaxString;
	state						: INT:=0;
	s_Typecode					: T_MaxString;
	s_Typedescription			: T_MaxString;
	fb_TonDel					: TON;

END_VAR
VAR_IN_OUT
	sVisu : sTDHandler;
END_VAR
VAR_INPUT
	TDActivationAlowed			: BOOL; (* Typedata activation alowed *)
END_VAR
VAR_OUTPUT
	DownLoadTime				: STRING;
END_VAR
info();
DisableTD();
IF 	NOT FirstCycle THEN
	IF	MP.sLastTDfile <> '' AND
		MP_TDPathLocal <> '' THEN
		FileNameRead 		:= CONCAT(MP_TDPathLocal,MP.sLastTDfile);
		FileReadTarget		:= '.TD';
		s_Xpath:='/dataentry/TD';
		ReadXML.bExecute	:=TRUE;
		FirstCycle:=TRUE;
	END_IF
END_IF

IF TD.TypeName <> TypeNameCopy THEN
	TypeNameCopy:=TD.TypeName;
	fb_ExpActTDNo.Start:=TRUE;
	MP.ST02.Override_Band:=TD.Override_Band;
	MP.ST00.Override:=TD.Override_Robi;
END_IF

IF 	FIND(sVisu.FileFilter,'*')= 0 THEN
	sVisu.FileFilter:=CONCAT(sVisu.FileFilter,'*');
END_IF

FileNameSearch := CONCAT(MP_TDPathLocal,sVisu.FileFilter);
FileNameSearch := CONCAT(FileNameSearch,MP_TDFileExtension);

fb_rTrigFilList(CLK:=CurrentVisu = 'TD_MAIN' );
IF 	FileIndexOld <> sTDHandler.FileIndex OR
	fb_rTrigFilList.Q OR
	FileFilterOld<>sVisu.FileFilter  THEN
	FileIndexOld:= sTDHandler.FileIndex;
	sVisu.FileListUpdate:=TRUE;
	FileFilterOld:=sVisu.FileFilter;
END_IF


(* --------------------------------------------------------------- *)
(* ------------------ Function Calls --------------------- *)
(* --------------------------------------------------------------- *)

FindFiles(
	bExecute			:=sVisu.FileListUpdate,
	sNetId				:= '',
	sPathName			:= FileNameSearch,
	pFindList			:= ADR(filesList),
	cbFindList		:= SIZEOF(filesList) ,
	tTimeout			:= t#1s );

sVisu.FileListUpdate:=FALSE;

WriteXML(
	sNetId				:= '',
	nMode				:= XMLSRV_ADDMISSING,
	sSymName			:= FileWriteSource,
	sFilePath			:= FileNameWrite ,
	sXPath				:= '/dataentry/TD',
	tTimeout			:= t#10s
 );

IF 	NOT WriteXML.bBusy OR WriteXML.bError THEN

	IF 	WriteXML.bExecute THEN
		sVisu.FileListUpdate:=TRUE;
	END_IF
	WriteXML.bExecute:=FALSE;

END_IF

ReadXML(
	sNetId				:= '',
	nMode				:= XMLSRV_SKIPMISSING ,
	sSymName			:= FileReadTarget,
	sFilePath			:= FileNameRead,
	sXPath				:= s_Xpath,				(* '/dataentry/TD',*)
	tTimeout			:= t#15s
 );


IF 	NOT ReadXML.bBusy AND
	ReadXML.bExecute	 THEN
	IF	FileReadTarget = '.TD' AND
		FileNameRead <>'' THEN
		lastTDActivate:=FileNameRead;
	END_IF
	TDValid:=TRUE;
END_IF

IF 	NOT ReadXML.bBusy OR
	ReadXML.bError THEN
	ReadXML.bExecute:=FALSE;
END_IF

j:=1;
FOR i:=1 TO NO_OF_FILES DO
	IF 	filesList[i].sFileName<>'' THEN
		sVisu.FileList[j]:=filesList[i].sFileName;
		j:=j+1;
	ELSE
		sVisu.FileList[j]:='';
		j:=j+1;
	END_IF
END_FOR

(* --------------------------------------------------------------- *)
(* -----------------  Visu interface ----------------------------- *)
(* --------------------------------------------------------------- *)
IF 	sVisu.FileIndex = 0 THEN
	sVisu.FileIndex:=1;
END_IF
sVisu.FileNameSelected:=sVisu.FileList[sVisu.FileIndex];

BtnActivate(
	Enable			:= sVisu.FileNameSelected <> MP.sLastTDfile AND sVisu.FileNameSelected <>'' AND ModeSelect.Mode <= MODE_MANUAL,
	Visible			:= TRUE,
	TextOn			:= 'Activate',
	TextOff			:= 'Activate',
	Button			:= sVisu.BtnActivate
  );

IF 	BtnActivate.PressedFlag THEN
	TD:=TDempty;
	TDCopy:=TDempty;
	FileNameRead 		:= CONCAT(MP_TDPathLocal,sVisu.FileNameSelected);
	FileReadTarget		:= '.TD';
	ReadXML.bExecute	:=TRUE;
	SetActivate			:=TRUE;
	gTypeDataValid 		:= FALSE;
	s_Xpath:='/dataentry/TD';
	MP.sLastTDfile		:=sVisu.FileNameSelected;
END_IF


IF 	SetActivate AND
	ModeSelect.Mode <= MODE_MANUAL OR gTInfo_FirstStart THEN

	IF 	NOT ReadXML.bBusy AND NOT ReadXML.bError THEN
		DownLoadTime:=gVarStrSystemTime;
		SetActivate:=FALSE;
		gTypeDataValid:=TRUE;
	ELSIF
		ReadXML.bBusy AND ReadXML.bError THEN
		SetActivate:=FALSE;
	END_IF
ELSIF
	ModeSelect.Mode<>MODE_MANUAL THEN
	SetActivate:=FALSE;
	(*ST00_LoadTInfo.Start:=FALSE;*)
END_IF
sVisu.TypeDataValid:=gTypeDataValid;


(*Automatisch sichern*)
IF	(MEMCMP(ADR(TDCopy), ADR(TD), SIZEOF(TDCopy)) <> 0 ) AND
	lastTDActivate<> '' AND
	NOT ReadXML.bBusy AND
	NOT ReadXML.bError THEN
	FileNameWrite	:= lastTDActivate;
	FileWriteSource	:= '.TD';
	WriteXML.bExecute:=TRUE;
END_IF
TDCopy:=TD;
TD.TypeName	:= MP.sLastTDfile;

(*============================*)

BtnSaveAs(
	Enable			:= sVisu.FileNameSelected = MP.sLastTDfile AND CurrentUserLevel >=6,
	Visible			:= TRUE ,
	TextOn			:= 'SaveAs',
	TextOff			:= 'SaveAs',
	Button			:= sVisu.BtnSaveAs
  );

IF 	BtnSaveAs.PressedFlag THEN
	b_Dialog_save_as_on:=TRUE;
END_IF

IF 	sVisu.FileNameSaveAs <>'' THEN
	FileNameWrite	:= CONCAT(MP_TDPathLocal,sVisu.FileNameSaveAs);
	FileNameWrite	:= CONCAT(FileNameWrite,MP_TDFileExtension);
  	TD.TypeName	:= sVisu.FileNameSaveAs;

	FileWriteSource	:= '.TD';
	WriteXML.bExecute:=TRUE;

	sVisu.FileNameSaveAs:='';
	b_Dialog_save_as_on:=FALSE;

END_IF

BtnDelete(
	Enable			:= sVisu.FileNameSelected <> MP.sLastTDfile AND sVisu.FileNameSelected<>'' AND CurrentUserLevel >=6,
	Visible			:= TRUE ,
(*	Enable			:= sVisu.FileNameSelected<>'',
	Visible			:= sVisu.FileNameSelected<>'',*)
	TextOn			:= 'Del',
	TextOff			:= 'Del',
	Button			:= sVisu.BtnDelete
  );


IF 	BtnDelete.PressedFlag THEN
	FileNameDelete 		:= CONCAT(MP_TDPathLocal,sVisu.FileNameSelected);
	DeleteXML.bExecute:=TRUE;
END_IF

DeleteXML(
	sNetId			:= '',
	sPathName		:= FileNameDelete,
	tTimeout		:= t#10s
 );
IF 	DeleteXML.bExecute AND
	DeleteXML.bBusy THEN
	DeleteXMLactive:=TRUE;
END_IF

IF 	DeleteXMLactive AND
	(NOT DeleteXML.bBusy OR  DeleteXML.bError) THEN
	sVisu.FileListUpdate:=TRUE;
	DeleteXMLactive:=FALSE;
END_IF


DeleteXML.bExecute:=FALSE;

(*send to ErrorHandler (to show Error-Line and to add into ErrorLogFile) *)
IF 	NOT TDValid THEN
	ErrorElapsed(CLK:= Error.Text<>''AND gVarDTSystemtime<> ErrorHandler.EmptyError.DateTime);
	IF 	ErrorElapsed.Q THEN
		Error.DateTime:=
		gVarDTSystemtime;
	END_IF
	Error.Text	:= 'TD: NOT valid';
	Error.No		:= 1;
	Error.Typ	:= 0;			(* 0=red 1:=orange 2:=blue *)
	ErrorHandler.AddError
				(ErrorToAdd	:=Error,
				sVisu		:=Visu.ErrorHandler);
END_IF

IF	TDValid AND
	FileNameReadCopy<> FileNameRead THEN
	Error.Text		:= CONCAT('TD: open ',FileNameRead);
	Error.DateTime	:=gVarDTSystemtime;
	Error.No			:= 1;
	Error.Typ		:= 0;			(* 0=red 1:=orange 2:=blue *)
	ErrorHandler.AddError
				(ErrorToAdd	:=Error,
				sVisu		:=Visu.ErrorHandler);

	FileNameReadCopy:=FileNameRead;
END_IF

IF	TDValid AND
	WriteXML.bExecute THEN
	Error.Text		:= CONCAT('TD: save ',FileNameWrite);
	Error.DateTime	:=gVarDTSystemtime;
	Error.No			:= 1;
	Error.Typ		:= 0;			(* 0=red 1:=orange 2:=blue *)
	ErrorHandler.AddError
				(ErrorToAdd	:=Error,
				sVisu		:=Visu.ErrorHandler);

END_IF

fb_ExpActTDNo(
	Start:= ,
	ExportStr:=TypeNameCopy ,
	FileName:= 'ActTD.txt',
	Path:=  s_tools_path,
	Mode:=FOPEN_MODEWRITE,
	Busy=> ,
	Done=> ,
	Error=> ,
	ErrorMsg=> );
END_PROGRAM
ACTION DisableTD:
(* Sperre der Typdateneingabe *)
gDisableTD := FALSE;
IF 	CurrentUserLevel <6  OR
	ModeSelect.Mode >  MODE_MANUAL THEN
	gDisableTD := TRUE;
END_IF
END_ACTION
ACTION Info:
(*immer wenn ein neu Datei ausgewhält wird, dann wird die Beschreibung und der Projektcode ausgelesen*)
fb_TonDel(PT:=t#20s);

IF 	FileIndexOld <> sTDHandler.FileIndex THEN
	fb_TonDel.IN:=FALSE;
	state:=5;
END_IF


CASE state OF
0:
	IF	fb_TonDel.Q THEN
		fb_TonDel.IN:=FALSE;
		s_Typecode:='';
		s_Typedescription:='';
	END_IF

5:
	IF 	FileIndexOld = sTDHandler.FileIndex AND
		NOT FindFiles.bBusy THEN
		state:=10;
	END_IF

10:
	FileNameRead 		:= CONCAT(MP_TDPathLocal,filesList[FileIndexOld].sFileName);
	FileReadTarget		:= 'TDHandler.s_Typecode';
	s_Xpath				:='/dataentry/TD/TYPECODE';
	ReadXML.bExecute	:=TRUE;
	IF	ReadXML.bBusy THEN
		state:=20;
		ReadXML.bExecute	:=FALSE;
	END_IF

20:
	IF	NOT ReadXML.bBusy AND
		NOT ReadXML.bError THEN
		state:=30;
	END_IF

30:
	FileNameRead 		:= CONCAT(MP_TDPathLocal,sVisu.FileNameSelected);
	FileReadTarget		:= 'TDHandler.s_Typedescription';
	s_Xpath				:='/dataentry/TD/TYPEDESCRIPTION';
	ReadXML.bExecute	:=TRUE;
	IF	ReadXML.bBusy THEN
		ReadXML.bExecute	:=FALSE;
		state:=40;
	END_IF

40:
	IF	NOT ReadXML.bBusy AND
		NOT ReadXML.bError THEN
		state:=0;
		fb_TonDel.IN:=TRUE;
	END_IF
END_CASE
END_ACTION

(* POU zLibrary/ept/Funktionsbausteine/FB_ExporString, ST *)
FUNCTION_BLOCK FB_ExporString
VAR_INPUT
	Start				:BOOL;
	ExportStr			:STRING(255);
	FileName		:STRING(255);
	Path				:STRING(255);
	Mode			:DWORD;
END_VAR
VAR_OUTPUT
	Busy				:BOOL;
	Done				:BOOL;
	Error				:BOOL;
	ErrorMsg			:STRING(255);

END_VAR
VAR
	fb_state_entry		:ST_StateEntry;
	nErrId				:UDINT;

	fbFileOpen			:FB_FileOpen;
	fbFilePuts			:FB_FilePuts;
	fbFileClose			:FB_FileClose;

	hFile				:UINT;

END_VAR

VAR CONSTANT
	Zeilenumbruch		:STRING:='$R$N';
END_VAR
(*======================================================
   PRG: FB_ExportString
 ------------------------------------------------------
   Auth: 		Werner Friedl    						 
   Date: 		30.10.2014    						     
   Rev.: 		1.0	
   Desc:		
		
   Historie:   1.0

 ========================================================*)
fb_state_entry(i16_pos:= 1);

CASE fb_state_entry.i16_step OF

0:	(*Objekt initialisieren*)
	fb_state_entry.i16_next_step:=INIT;

10:	(*initialisieren*)
	fb_state_entry.i16_next_step:=BEREIT;

BEREIT:(*Start*)

	IF	Start THEN  (*initialisieren*)
		Start:=FALSE;
		Busy:=TRUE;
		Error:=FALSE;
		Done:=FALSE;
		nErrId:=0;
		ErrorMsg:='';
		fb_state_entry.i16_next_step:=110;

	END_IF

110: (*Datei erstellen*)

	FileName:=CONCAT(Path,FileName);

	fbFileOpen.sPathName:=FileName;
 	fbFileOpen.bExecute:=TRUE;

	IF 	NOT fbFileOpen.bBusy   THEN
		fb_state_entry.i16_next_step:=120;
	END_IF

120: (*Datei erstellen*)

	IF 	NOT fbFileOpen.bBusy THEN
		fbFileOpen.bExecute:=FALSE;
		IF 	fbFileOpen.bError THEN
			nErrId:=fbFileOpen.nErrId;
			fb_state_entry.i16_next_step:=FEHLER;
			ErrorMsg:='Fehler beim Öffnen der Datei';
		ELSE
			fb_state_entry.i16_next_step:=130;
		END_IF
	END_IF

130: (*String in Datei eintragen*)
	IF fb_state_entry.E THEN
		;
	END_IF

	fbFilePuts.sLine:=CONCAT(ExportStr,Zeilenumbruch);
	fbFilePuts.bExecute:=TRUE;

	IF  fbFilePuts.bBusy THEN
		fb_state_entry.i16_next_step:=140;
	END_IF

140: (*String in Datei eintragen*)

	IF 	NOT fbFilePuts.bBusy THEN
		fbFilePuts.bExecute:=FALSE;
		IF 	fbFilePuts.bError THEN
			nErrId:=fbFilePuts.nErrId;
			fb_state_entry.i16_next_step:=150;
			ErrorMsg:='Fehler beim String Eintragen in der Datei';
			Error:=TRUE;
		ELSE
			fb_state_entry.i16_next_step:=150;
		END_IF
	END_IF

150:(*Datei schließen*)

	fbFileClose.bExecute:=TRUE;
	IF 	fbFileClose.bBusy THEN
		fb_state_entry.i16_next_step:=160;
	END_IF

160:(*Datei schließen*)

	IF NOT fbFileClose.bBusy THEN
		fbFileClose.bExecute:=FALSE;
		IF 	fbFileClose.bError THEN
			nErrId:=fbFileClose.nErrId;
			ErrorMsg:='Fehler beim Schließen der Datei';
			Error:=TRUE;
		ELSE
			fb_state_entry.i16_next_step:=170;
		END_IF
	END_IF

	IF	Error THEN
		fb_state_entry.i16_next_step:=FEHLER;
	END_IF

170: (*fertig*)
	Busy:=FALSE;
	Done:=TRUE;
	fb_state_entry.i16_next_step:=10;

FEHLER: (*Fehler*)
	fb_state_entry.i16_next_step:=10;
	Busy:=FALSE;
	Error:=TRUE;
END_CASE

fb_state_entry(i16_pos:= 2 );

fbFileOpen(
	sNetId:='',
	sPathName:= ,
	nMode:=mode,
	ePath:=PATH_GENERIC,
	bExecute:= ,
	tTimeout:=T#1s,
	hFile=> hFile);

fbFilePuts(
	sNetId:='',
	hFile:=hFile,
	sLine:= ,
	bExecute:= ,
	tTimeout:=t#1s);

fbFileClose(
	sNetId:='',
	hFile:=hFile,
	bExecute:= ,
	tTimeout:=t#1s);
END_FUNCTION_BLOCK

(* POU System/MPHandler/MPHandler, ST *)
PROGRAM MPHandler
VAR

	LocalFiles					: FB_EnumFindFileList;
	ExportFiles					: FB_EnumFindFileList;

	CreateDirectory			:FB_CreateDir;

	CopyFiles						:	FB_FileCopy;

	WriteXML						: FB_XmlSrvWriteByName;
	ReadXML							: FB_XmlSrvReadByName;


	LocalDirectory					: ARRAY[1..200] OF ST_FindFileEntry;
	ExportDirectory				: ARRAY[1..200] OF ST_FindFileEntry;

	i										:	DINT;
	j										:	DINT;

	FileNameSearchExport		:	STRING(255);
	FileNameSearchLocal		:	STRING(255);

	FileListUpdateExport		:	BOOL;
	FileListUpdateLocal		:	BOOL;

	BtnImport							:	VisuButton;
	BtnExport							:	VisuButton;


	StepExport					:	DINT;

	Delay : TON;

	NoOfTDFilesToCopy	:	DINT;
	AktFileToCopy			:	DINT;

	TempStringSource	:	STRING;
	TempStringTarget	:	STRING;

	Backslash						:	STRING :='\';

	MP_BAK							: sMachPara;
END_VAR
VAR_IN_OUT
	sVisu : sMPHandler;
END_VAR
DisableMP();
j:=1;
FOR i:=1 TO 20 DO
	IF ExportDirectory[i].sFileName<>''
	THEN
		sVisu.FileListExport[j]:=ExportDirectory[i].sFileName;
		j:=j+1;
	ELSE
		sVisu.FileListExport[j]:='';
		j:=j+1;
	END_IF
END_FOR
j:=1;
FOR i:=1 TO 20 DO
	IF LocalDirectory[i].sFileName<>''
	THEN
		sVisu.FileListLocal[j]:=LocalDirectory[i].sFileName;
		j:=j+1;
	ELSE
		sVisu.FileListLocal[j]:='';
		j:=j+1;
	END_IF
END_FOR


(* --------------------------------------------------------------- *)
(* -----------------  sVisu interface ----------------------------- *)
(* --------------------------------------------------------------- *)



BtnImport(
	Enable			:= StepExport=0,
	Visible			:= FALSE,
	TextOn			:= 'Import',
	TextOff			:= 'Import',
	Button			:= sVisu.BtnImport
  );



BtnExport(
	Enable			:= StepExport=0,
	Visible			:= TRUE,
	TextOn			:= 'Export',
	TextOff			:= 'Export',
	Button			:= sVisu.BtnExport
  );

IF BtnExport.PressedFlag
THEN
StepExport:=1;

END_IF


CASE StepExport OF
(* Überprüfen ob Laufwerk vorh. ist *)
	0:	sVisu.MessageString:='';
	1:	FileNameSearchExport	:=	MP_ExportDrive;
			sVisu.MessageString:='';
			StepExport			:=	2(*2*);
	2:	FileListUpdateExport:=TRUE;
			StepExport			:=	3;
	3:	IF ExportFiles.bError OR (ExportFiles.bEOE AND ExportFiles.nFindFiles=0 AND NOT ExportFiles.bBusy)
			THEN
				sVisu.MessageString:='Exportlaufwerk wurde nichterkannt!';
				FileListUpdateExport:=FALSE;
				StepExport			:=	999;
			ELSIF ExportFiles.bEOE AND  ExportFiles.nFindFiles>0
			THEN
				FileListUpdateExport:=FALSE;
				StepExport			:=	4;
			END_IF
	4:	IF NOT ExportFiles.bBusy
			THEN
				StepExport			:=	10;
			END_IF
(* Typdaten Exportpfad prüfen / anlegen *)
	10:	FileNameSearchExport	:=	MP_ExportDrivePathTD;(* 4 *)
			sVisu.MessageString:='';
			StepExport			:=	11;
	11:	FileListUpdateExport:=TRUE;
			StepExport			:=	12;
	12:	IF ExportFiles.nFindFiles=0 AND (ExportFiles.bEOE OR ExportFiles.bError)
			THEN
				sVisu.MessageString:='Typdatenpfad wird angelegt! -> /_TD/';
				FileListUpdateExport:=FALSE;
				StepExport			:=	13;
			ELSIF ExportFiles.nFindFiles>0 AND (ExportFiles.bEOE OR ExportFiles.bError)
			THEN
				FileListUpdateExport:=FALSE;
				StepExport			:=	20;
			END_IF
	13:	CreateDirectory.sPathName:=MP_ExportDrivePathTD;
			CreateDirectory.bExecute:=FALSE;
			StepExport			:=	14;
	14:	CreateDirectory.bExecute:=TRUE;
			IF CreateDirectory.bBusy
			THEN
				StepExport			:=	15;
			END_IF
	15:	IF NOT CreateDirectory.bBusy AND NOT CreateDirectory.bError
			THEN
				StepExport			:=	20;

			ELSIF NOT CreateDirectory.bBusy AND CreateDirectory.bError
			THEN
				StepExport			:=	999;
				sVisu.MessageString:='Fehler bein erstellen des Typdatenpfades';
			END_IF


(* Maschinenparameter Exportpfad prüfen / anlegen *)
	20:	FileNameSearchExport	:=	MP_ExportDrivePathMP;
			sVisu.MessageString:='';
			StepExport			:=	21;
	21:	FileListUpdateExport:=TRUE;
			StepExport			:=	22;
	22:	IF ExportFiles.nFindFiles=0 AND (ExportFiles.bEOE OR ExportFiles.bError)
			THEN
				sVisu.MessageString:='Maschinenparameterpfad  wird angelegt! -> /_MP/';
				FileListUpdateExport:=FALSE;
				StepExport			:=	23;
			ELSIF ExportFiles.nFindFiles>0 AND (ExportFiles.bEOE OR ExportFiles.bError)
			THEN
				FileListUpdateExport:=FALSE;
				StepExport			:=	40;
			END_IF
	23:	CreateDirectory.sPathName:=MP_ExportDrivePathMP;
			CreateDirectory.bExecute:=FALSE;
			StepExport			:=	24;
	24:	CreateDirectory.bExecute:=TRUE;
			IF CreateDirectory.bBusy
			THEN
				StepExport			:=	25;
			END_IF
	25:	IF NOT CreateDirectory.bBusy AND NOT CreateDirectory.bError
			THEN
				StepExport			:=	40;

			ELSIF NOT CreateDirectory.bBusy AND CreateDirectory.bError
			THEN
				StepExport			:=	999;
				sVisu.MessageString:='Fehler bein erstellen des Maschinenparameterpfades';
			END_IF

	(* Typdaten kopieren *)
	40: sVisu.MessageString:='';
			StepExport			:=	41;
			FileNameSearchExport	:=	CONCAT(CONCAT(MP_ExportDrivePathTD,Backslash),MP_TDSearchString);
			FileNameSearchLocal		:=	CONCAT(MP_TDPathLocal,MP_TDSearchString);
	41: FileListUpdateExport:=TRUE;
			StepExport			:=	42;
	42: IF ExportFiles.bEOE OR ExportFiles.bError
			THEN
				FileListUpdateExport:=FALSE;
				StepExport			:=	43;
			END_IF
	43: FileListUpdateLocal:=TRUE;
			StepExport			:=	44;
	44: IF LocalFiles.nFindFiles=0 AND (LocalFiles.bEOE OR LocalFiles.bError)
			THEN
				sVisu.MessageString:='Es wurden keine Typdaten zum Exportieren gefunden!';
				FileListUpdateLocal:=FALSE;
				StepExport			:=	100;
			ELSIF LocalFiles.nFindFiles>0 AND (LocalFiles.bEOE OR LocalFiles.bError)
			THEN
				FileListUpdateLocal:=FALSE;
				NoOfTDFilesToCopy:=LocalFiles.nFindFiles;
				StepExport			:=	60;
			END_IF

	60:	AktFileToCopy		:=	1;
			StepExport			:=	61;

	61: (* Set Path *)
			TempStringSource					:=	CONCAT(MP_TDPathLocal,LocalDirectory[AktFileToCopy].sFileName);
			TempStringTarget					:=	CONCAT(CONCAT(MP_ExportDrivePathTD,Backslash),LocalDirectory[AktFileToCopy].sFileName);
			CopyFiles.srcFileName			:=	TempStringSource;
			CopyFiles.destFileName		:=	TempStringTarget;
			CopyFiles.bExecute				:=	FALSE;
			StepExport								:=	62;
			sVisu.MessageString:='Typdaten werden kopiert...';

	62: (* Start to Copy *)
			CopyFiles.bExecute				:=	TRUE;
			IF CopyFiles.bBusy
			THEN
				StepExport								:=	63;
			END_IF
	63: (* Copy Done *)
			CopyFiles.bExecute				:=	FALSE;
			IF NOT CopyFiles.bBusy AND NOT CopyFiles.bError
			THEN
				StepExport								:=	64;
			ELSIF NOT CopyFiles.bBusy AND CopyFiles.bError
			THEN
				StepExport								:=	999;
				sVisu.MessageString:='Fehler beim kopieren der Typdaten!';
			END_IF
	64: FileListUpdateExport:=TRUE;
			StepExport			:=	65;
	65:	(* Check last file To copy *)
			FileListUpdateExport:=FALSE;
			IF AktFileToCopy>=NoOfTDFilesToCopy
			THEN
				StepExport								:=	66;
			ELSE
				AktFileToCopy							:=	AktFileToCopy + 1;
				StepExport								:=	61;
			END_IF

	66:	(* All Files copied *)
			sVisu.MessageString:='Typdaten kopieren abgeschlossen!';
				StepExport								:=	100;

 100:	(* Maschinendaten sichern *)
			WriteXML.bExecute					:=	FALSE;
			StepExport								:=	101;
 101: WriteXML.bExecute					:=	TRUE;
			IF WriteXML.bBusy
			THEN
				WriteXML.bExecute					:=	FALSE;
				StepExport								:=	102;
			END_IF
 102: IF NOT WriteXML.bBusy AND NOT WriteXML.bError
			THEN
				WriteXML.bExecute					:=	FALSE;
				StepExport								:=	110;
			ELSIF NOT WriteXML.bBusy AND WriteXML.bError
			THEN
				sVisu.MessageString:='Fehler bein schreiben der XML-Datei für die Maschinenparameter....';
				WriteXML.bExecute					:=	FALSE;
				StepExport								:=	999;
			END_IF
 110:
			(* Set Path *)
			TempStringSource					:=	CONCAT(CONCAT(MP_ExportDrivePathMP, Backslash),MP_MPExportFilename);(*'\Hard Disk\_MP\MachPara.xml';*)
			TempStringTarget					:=	CONCAT(CONCAT(MP_ExportDrivePathMP, Backslash),MP_MPExportFilename);(*'\Hard Disk2\_MP\MachPara.xml';*)
			CopyFiles.srcFileName			:=	TempStringSource;
			CopyFiles.destFileName		:=	TempStringTarget;
			CopyFiles.bExecute				:=	FALSE;
			StepExport								:=	111;
			sVisu.MessageString:='Maschinenparameter werden kopiert...';

	111: (* Start to Copy *)
			CopyFiles.bExecute				:=	TRUE;
			IF CopyFiles.bBusy
			THEN
				StepExport								:=	112;
			END_IF
	112: (* Copy Done *)
			CopyFiles.bExecute				:=	FALSE;
			IF NOT CopyFiles.bBusy AND NOT CopyFiles.bError
			THEN
				sVisu.MessageString:='Maschinenparameter kopieren abgeschlossen!';
				StepExport								:=	999;
			ELSIF NOT CopyFiles.bBusy AND CopyFiles.bError
			THEN
				StepExport								:=	999;
				sVisu.MessageString:='Fehler beim kopieren der Maschinenparameter!';
			END_IF
 999:	Delay(IN:= FALSE, PT:= t#0s);
			StepExport			:=	1000;
1000: Delay(IN:= TRUE, PT:= t#1s);
			IF delay.Q
			THEN
				StepExport			:=	0;
			END_IF
END_CASE


ExportFiles(
	bExecute			:=sVisu.FileListUpdate OR FileListUpdateExport,
	sNetId				:= '',
	sPathName			:= FileNameSearchExport,
	pFindList			:= ADR(ExportDirectory),
	cbFindList		:= SIZEOF(ExportDirectory) ,
	tTimeout			:= t#10s );

LocalFiles(
	bExecute			:=sVisu.FileListUpdate OR FileListUpdateLocal,
	sNetId				:= '',
	sPathName			:= FileNameSearchLocal,
	pFindList			:= ADR(LocalDirectory),
	cbFindList		:= SIZEOF(LocalDirectory) ,
	tTimeout			:= t#1s );

CopyFiles(
	srcNetId:= '',
	destNetId:= '',
	tAdsSTATE_TIMEOUT:= t#1s);


WriteXML(
	sNetId				:= '',
	nMode					:= XMLSRV_ADDMISSING,
 	sSymName				:='.MP',
	sFilePath			:= CONCAT(CONCAT(MP_ExportDrivePathMP, Backslash),MP_MPExportFilename),
	sXPath				:= '/dataentry/MP',
	tTimeout			:= t#10s );


sVisu.FileListUpdate:=FALSE;

CreateDirectory(
	sNetId:= '' );


ReadXML(
	sNetId:= '',
	nMode:= XMLSRV_ADDMISSING,
	sSymName:= '.MP',
	sFilePath:= '\Hard Disk\_MP\MachPara.xml',
	sXPath:= '/dataentry/MP'
);


IF MEMCMP(ADR(MP),ADR(MP_BAK),SIZEOF(MP_BAK))<>0
THEN
	Visu.SavePersistentData:=TRUE;
	MP_BAK:=MP;
END_IF
END_PROGRAM
ACTION DisableMP:
(* Sperre der Typdateneingabe *)
gDisableMP := FALSE;
IF 	CurrentUserLevel <6  OR
	ModeSelect.Mode > MODE_MANUAL THEN
	gDisableMP := TRUE;
END_IF
END_ACTION

(* POU System/HelpFunctions/FB_FileCopy, ST *)
FUNCTION_BLOCK FB_FileCopy
VAR_INPUT
	srcNetId				: T_AmsNetId;	(* TwinCAT network address of the source file *)
	srcFileName				: T_MaxString;	(* source file path and name *)
	destNetId				: T_AmsNetId;	(* TwinCAT network address of the destination file *)
	destFileName			: T_MaxString;  	(* destination file path and name *)
	bExecute				: BOOL;		(* rising edge starts fb execution *)
	tAdsSTATE_TIMEOUT	: TIME;		(* ads STATE_TIMEOUT *)
END_VAR
VAR_OUTPUT
	bBusy		  		:BOOL;
	bError				:BOOL;
	nErrId				:UDINT;
END_VAR
VAR
	fbFileOpen			:FB_FileOpen;
	fbFileClose			:FB_FileClose;
	fbFileRead			:FB_FileRead;
	fbFileWrite			:FB_FileWrite;

	hSrcFile				:UINT	:= 0;(* file handle of the source file *)
	hDestFile			:UINT	:= 0;(* file handle of the destination file *)

	Step				:DWORD;
	RisingEdge			:R_TRIG;

	buffRead			:ARRAY[1..100000] OF BYTE;(* buffer *)
	cbReadLength		:UDINT:=0;
END_VAR
RisingEdge(CLK:=bExecute);
IF RisingEdge.Q THEN
	IF 	NOT bBusy THEN
		bBusy := TRUE;
		bError:= FALSE;
		nErrId:=0;
		Step := 1;
		cbReadLength:=0;
		hSrcFile:=0;
		hDestFile:=0;
	END_IF
END_IF


CASE Step OF
	0:(* do nothing *)
	;

	1:(* open source file *)
	fbFileOpen(  bExecute := FALSE  );
	fbFileOpen(	sNetId := srcNetId,
		sPathName := srcFileName,
		nMode := FOPEN_MODEREAD OR FOPEN_MODETEXT ,
		ePath := PATH_GENERIC,
		tTimeout := tAdsSTATE_TIMEOUT,
		bExecute := TRUE );
		Step := Step + 1;

	2:
	fbFileOpen( bExecute := FALSE );
	IF ( NOT fbFileOpen.bBusy ) THEN
		IF ( fbFileOpen.bError ) THEN
			nErrId := fbFileOpen.nErrId;
			bError := TRUE;
			Step := 50;
		ELSE
			hSrcFile := fbFileOpen.hFile;
			Step := Step + 1;
		END_IF
	END_IF

	3:(* open destination file *)
	fbFileOpen(  bExecute := FALSE  );
	fbFileOpen( 	sNetId := destNetId,
			sPathName := destFileName,
			nMode := FOPEN_MODEWRITE OR FOPEN_MODETEXT ,
			ePath := PATH_GENERIC,
			tTimeout := tAdsSTATE_TIMEOUT,
			bExecute := TRUE );
	Step := Step+1;

	4:
	fbFileOpen(  bExecute := FALSE  );
	IF ( NOT fbFileOpen.bBusy ) THEN
		IF ( fbFileOpen.bError ) THEN
			nErrId := fbFileOpen.nErrId;
			bError := TRUE;
			Step := 50;
		ELSE
			hDestFile := fbFileOpen.hFile;
			Step := Step + 1;
		END_IF
	END_IF

	5:(*read data from source file*)
	cbReadLength := 0;
	fbFileRead( bExecute:= FALSE );
	fbFileRead( 	sNetId:=SrcNetId,
			hFile:=hSrcFile,
			pReadBuff:= ADR(buffRead),
			cbReadLen:= SIZEOF(buffRead),
			bExecute:=TRUE,
			tTimeout:=tAdsSTATE_TIMEOUT );
	Step := Step + 1;

	6:
	fbFileRead( bExecute:= FALSE );
	IF ( NOT fbFileRead.bBusy ) THEN
		IF ( fbFileRead.bError ) THEN
			nErrId := fbFileRead.nErrId;
			bError := TRUE;
			Step := 50;
		ELSE
			cbReadLength := fbFileRead.cbRead;
			Step := Step + 1;
		END_IF
	END_IF

	7:(*write data to destination file*)
	fbFileWrite( bExecute := FALSE );
	fbFileWrite(	sNetId:=DestNetId,
			hFile:=hDestFile,
			pWriteBuff:= ADR(buffRead),
			cbWriteLen:= cbReadLength,
			bExecute:=TRUE,
			tTimeout:=tAdsSTATE_TIMEOUT );
	Step := Step + 1;

	8:
	fbFileWrite( bExecute := FALSE );
	IF ( NOT fbFileWrite.bBusy ) THEN
		IF ( fbFileWrite.bError ) THEN
			nErrId := fbFileWrite.nErrId;
			bError := TRUE;
			Step := 50;
		ELSE
			IF fbFileRead.bEOF THEN (*Check if the EOF flag ist set *)
				Step := 50;(*cleanup: close the destination and source files *)
			ELSE
				Step := 5; (* repeat reading *)
			END_IF
		END_IF
	END_IF

	30:(* close the destination file *)
	fbFileClose( bExecute := FALSE );
	fbFileClose( 	sNetId:=destNetId,
			hFile:=hDestFile,
			bExecute:=TRUE,
			tTimeout:=tAdsSTATE_TIMEOUT );
	Step := Step + 1;

	31:
	fbFileClose( bExecute := FALSE );
	IF ( NOT fbFileClose.bBusy ) THEN
		IF ( fbFileClose.bError ) THEN
			nErrId := fbFileClose.nErrId;
			bError := TRUE;
		END_IF
		Step := 50;
		hDestFile := 0;
	END_IF

	40: (* close source file *)
	fbFileClose( bExecute := FALSE );
	fbFileClose( 	sNetId:=srcNetId,
			hFile:=hSrcFile,
			bExecute:=TRUE,
			tTimeout:=tAdsSTATE_TIMEOUT );
	Step := Step + 1;

	41:
	fbFileClose( bExecute := FALSE );
	IF ( NOT fbFileClose.bBusy ) THEN
		IF ( fbFileClose.bError ) THEN
			nErrId := fbFileClose.nErrId;
			bError := TRUE;
		END_IF
		Step := 50;
		hSrcFile := 0;
	END_IF

	50: (*error or ready => cleanup*)
	IF ( hDestFile <> 0 ) THEN
		Step := 30; (* close the destination file*)
	ELSIF (hSrcFile <> 0 ) THEN
		Step := 40; (* close the source file *)
	ELSE
		Step := 0;	(* ready *)
		bBusy := FALSE;
	END_IF

END_CASE
END_FUNCTION_BLOCK

(* POU System/MP_ShiftHandler/MP_ShiftHandler, ST *)
PROGRAM MP_ShiftHandler
VAR
	TodNow				: TOD;

	TempStartTOD 		: TOD;
	TempEndTOD 			: TOD;

	TempNightShift		: BOOL;

	TimeDayBegins		: TOD := TOD#00:00;
	TimeDayEnds			: TOD := TOD#23:59:59.999;

	NumberofShifts		: DINT;
	Idx					: DINT;

	NoShiftActive		: sMP_ShiftData;
	OneShiftIsActive	: BOOL;

END_VAR
NoShiftActive.ShiftIndex:=999;
NoShiftActive.ShiftName:='keine Schicht Activ';


NumberofShifts:=SIZEOF(MP.ShiftData.Shift)/SIZEOF(mp.ShiftData.ActiveShift);

TodNow:=DT_TO_TOD(SYSTEMTIME_TO_DT(gVarSystemtime));
TodNow:=	DINT_TO_TOD(TOD_TO_DINT(TodNow)	+	WORD_TO_DINT(gVarSystemtime.wMilliseconds));


OneShiftIsActive:=FALSE;

FOR Idx:=1 TO NumberofShifts DO


	MP.ShiftData.Shift[Idx].TimeStart.wYear:=gVarSystemtime.wYear;
	MP.ShiftData.Shift[Idx].TimeStart.wMonth:=gVarSystemtime.wMonth;
	MP.ShiftData.Shift[Idx].TimeStart.wDay:=gVarSystemtime.wDay;
	MP.ShiftData.Shift[Idx].TimeStart.wDayOfWeek:=gVarSystemtime.wDayOfWeek;
	MP.ShiftData.Shift[Idx].TimeStart.wSecond:=0;
	MP.ShiftData.Shift[Idx].TimeStart.wMilliseconds:=0;


	MP.ShiftData.Shift[Idx].TimeEnd.wYear:=gVarSystemtime.wYear;
	MP.ShiftData.Shift[Idx].TimeEnd.wMonth:=gVarSystemtime.wMonth;
	MP.ShiftData.Shift[Idx].TimeEnd.wDay:=gVarSystemtime.wDay;
	MP.ShiftData.Shift[Idx].TimeEnd.wDayOfWeek:=gVarSystemtime.wDayOfWeek;
	MP.ShiftData.Shift[Idx].TimeEnd.wSecond:=59;
	MP.ShiftData.Shift[Idx].TimeEnd.wMilliseconds:=0;


	TempStartTOD:=DT_TO_TOD(SYSTEMTIME_TO_DT(MP.ShiftData.Shift[Idx].TimeStart));

	TempStartTOD:=	DINT_TO_TOD(TOD_TO_DINT(TempStartTOD)	+	WORD_TO_DINT(MP.ShiftData.Shift[Idx].TimeStart.wMilliseconds));

	TempEndTOD:=DT_TO_TOD(SYSTEMTIME_TO_DT(MP.ShiftData.Shift[Idx].TimeEnd));

	MP.ShiftData.Shift[Idx].TimeEnd.wMilliseconds:=999;
	TempEndTOD:=	DINT_TO_TOD(TOD_TO_DINT(TempEndTOD)	+	WORD_TO_DINT(MP.ShiftData.Shift[Idx].TimeEnd.wMilliseconds));


	TempNightShift:=TOD_TO_DINT(TempStartTOD)>TOD_TO_DINT(TempEndTOD);

	IF 	NOT TempNightShift THEN
		MP.ShiftData.Shift[Idx].ShiftActive:=	(TodNow >= TempStartTOD)	AND (TodNow <= TempEndTOD);
	ELSE
		MP.ShiftData.Shift[Idx].ShiftActive:=	(TodNow >= TempStartTOD) AND
											(TodNow <= TimeDayEnds) OR (TodNow >= TimeDayBegins) AND
											(TodNow <= TempEndTOD);
	END_IF

	IF 	NOT OneShiftIsActive THEN
		OneShiftIsActive:=MP.ShiftData.Shift[Idx].ShiftActive;
		MP.ShiftData.ActiveShift:=MP.ShiftData.Shift[Idx];
	END_IF

END_FOR

IF 	NOT OneShiftIsActive THEN
	MP.ShiftData.ActiveShift:=NoShiftActive;
END_IF
END_PROGRAM

(* POU Stations/ST_00/ST00_FBs/_CallFBs, ST *)
PROGRAM _CallFBs


VAR



END_VAR
ST00_CallFBs();
ST03_CallFBs();

ST08_CallFBs();
END_PROGRAM

(* POU Stations/ST_00/ST00_FBs/ST00_CallFBs, ST *)
PROGRAM ST00_CallFBs
(*   Author:           *)


VAR



END_VAR
(* ----------------------------------------------------------------------------------------- *)
(* 																				Eingänge  																				 *)
(* ----------------------------------------------------------------------------------------- *)


(* Call ST00_40_F1 Vorsicherungen Leistung iO (DigIn) *)
ST00_40_F1(	sVisu:=Visu.ST00_40_F1,
			Reset:=gResetAll,
			CheckSignalHigh:=TRUE,
);

(* Call ST03_210_S1 Not-Aus 1 Anlage ausgelöst (DigIn) *)
ST03_210_S1(	sVisu:=Visu.ST03_210_S1,
				Reset:=gResetAll,
				CheckSignalLow:=TRUE,
);
(* Call ST08_210_S2 Not-Aus 2 Anlage ausgelöst (DigIn) *)
ST08_210_S2(	sVisu:=Visu.ST08_210_S2,
				Reset:=gResetAll,
				CheckSignalLow:=FALSE,
				CheckSignalHigh:=TRUE,
);

(* Call ST00_X4_16  Not-Halt 2 Tampondrucker  (DigIn) *)
ST00_X4_16(	sVisu:=Visu.ST00_X4_16,
			Reset:=gResetAll,
			CheckSignalLow:=TRUE,
);

(* Call ST00_200_A1_A1 Not-Aus iO (DigIn) *)
ST00_200_A1_A1(	sVisu:=Visu.ST00_200_A1_A1,
				Reset:=gResetAll,
				CheckSignalHigh:=TRUE,
);

(* Call ST00_220_S1 Schutztüre 1 geöffnet (DigIn) *)
ST00_220_S1(sVisu:=Visu.ST00_220_S1,
			Reset:=gResetAll,
			CheckSignalLow:=TRUE,
);

(* Call ST00_220_S2 Schutztüre 1 geöffnet (DigIn) *)
ST00_220_S2(sVisu:=Visu.ST00_220_S2,
			Reset:=gResetAll,
			CheckSignalLow:=TRUE,
);

(* Call ST00_230_S2_E1 Schutztüre 1 geschlossen (DigIn) *)
ST00_230_S2_E1(sVisu:=Visu.ST00_230_S2_E1,
			Reset:=gResetAll,
			(* CheckSignalHigh:=TRUE,*) (* @@@ *)
);

(* Call ST00_240_S1 Schutztüre 9 geschlossen (DigIn) *)
ST00_240_S1(sVisu:=Visu.ST00_240_S1,
			Reset:=gResetAll,
);

(* Call ST00_226_S1 Hubtüre 1 Schleuse Einlauf STN 8 geschlossen (DigIn) *)
ST00_226_S1(sVisu:=Visu.ST00_226_S1,
			Reset:=gResetAll,
);
(* Call ST00_226_S2 Hubtüre 2 Schleuse Einlauf STN 8 geschlossen (DigIn) *)
ST00_226_S2(sVisu:=Visu.ST00_226_S2,
			Reset:=gResetAll,
);
(* Call ST00_227_S1 Hubtüre 3 Schleuse Auslauf STN 8 geschlossen (DigIn) *)
ST00_227_S1(sVisu:=Visu.ST00_227_S1,
			Reset:=gResetAll,
);
(* Call ST00_227_S2 Hubtüre 4 Schleuse Auslauf STN 8 geschlossen (DigIn) *)
ST00_227_S2(sVisu:=Visu.ST00_227_S2,
			Reset:=gResetAll,
);
(* Call ST00_229_S1 Schutztüre Einlauf Tray STN 8 geschlossen (DigIn) *)
ST00_229_S1(sVisu:=Visu.ST00_229_S1,
			Reset:=gResetAll,
);
(* Call ST00_230_S1 Schutztüre Auslauf Tray STN 8 geschlossen (DigIn) *)
ST00_230_S1(sVisu:=Visu.ST00_230_S1,
			Reset:=gResetAll,
);
(* Call ST00_231_S1 Schutztüre Panel / Rutsche STN 8 geschlossen (DigIn) *)
ST00_231_S1(sVisu:=Visu.ST00_231_S1,
			Reset:=gResetAll,
);
(* Call ST00_232_S1 Schutztüre 8 Auslauf Tray STN 8 geschlossen (DigIn) *)
ST00_232_S1(sVisu:=Visu.ST00_232_S1,
			Reset:=gResetAll,
);
(* Call ST00_170Motorschutz Motorschutz in Ordnung (DigIn) *)
ST00_170_Motorschutz( sVisu:=Visu.ST00_170_Motorschutz,
						Reset:=gResetAll,
						CheckSignalHigh:=TRUE,
);

(* Call ST00_Thermokont Thermokontakt in Ordnung (DigIn) *)
ST00_170_Thermokont(	sVisu:=Visu.ST00_170_Thermokont,
						Reset:=gResetAll,
						CheckSignalHigh:=TRUE,
);


(* Call ST00_228_S1 Pallettierer in Position (DigIn) *)
ST00_228_S1(sVisu:=Visu.ST00_228_S1,
			Reset:=gResetAll,
);

(* Call ST00_71_X1_3 Schnittstelle Bedrucken Tinte JSK auf Übergabeposition (DigIn) *)
ST00_71_X1_3(sVisu:=Visu.ST00_71_X1_3,
			Reset:=gResetAll,
);

(* Call ST00_71_X1_4 Schnittstelle Bedrucken Tinte Druckstation betriebsbereit (DigIn) *)
ST00_71_X1_4(sVisu:=Visu.ST00_71_X1_4,
			Reset:=gResetAll,
);

(* Call ST00_72_X1_3 Schnittstelle Tampondrucker Teil in Abholposition (DigIn) *)(*Band Entnahmeposition 1*)
ST00_72_X1_3(sVisu:=Visu.ST00_72_X1_3,
			Reset:=gResetAll,
);

(* Call ST00_72_X1_8 Schnittstelle Tampondrucker Druck abgeschlossen (DigIn) *)
ST00_72_X1_8(sVisu:=Visu.ST00_72_X1_8,
			Reset:=gResetAll,
);

(* Call ST00_292_S1_STOP Bedienstelle Produktion Stop (DigIn) *)
ST00_292_S1_STOP(	sVisu:=Visu.ST00_292_S1_STOP,
					Reset:=gResetAll,
);
(* Call ST00_292_S2_START Bedienstelle Produktion Start (DigIn) *)
ST00_292_S2_START(	sVisu:=Visu.ST00_292_S2_START,
					Reset:=gResetAll,
);

(* Call ST00_292_S3_RESET Bedienstelle Produktion Start (DigIn) *)
ST00_292_S3_RESET(	sVisu:=Visu.ST00_292_S3_RESET,
					Reset:=gResetAll,
);
(* Call ST00_350_B20_0 Druckschalter Wartungseinheit Hauptluft min.6 bar (DigIn) *)
ST00_350_B20_0(	sVisu:=Visu.ST00_350_B20_0,
				Reset:=gResetAll,
				CheckSignalHigh:=TRUE,
);

(* Call 	ST00_245_V1			Verriegelung Schutztüren-Leuchte (DigOutIn) *)
ST00_245_V1(	sVisu:=Visu.ST00_245_V1,
					Reset:=gResetAll,
);

(* Call 	ST00_245_V2_START	Bedienstelle Start-Leuchte (DigOutIn) *)
ST00_245_V2_START(	sVisu:=Visu.ST00_245_V2_START,
					Reset:=gResetAll,
);

(* Call 	ST00_245_V3_RESET	Bedienstelle Reset-Schutztüren-Leuchte (DigOutIn) *)
ST00_245_V3_RESET(	sVisu:=Visu.ST00_245_V3_RESET,
					Reset:=gResetAll,
);

(* Call 	ST00_245_S1_STOP 	Bedienstelle Produktion Stop (DigIn) *)
ST00_245_S1_STOP(	sVisu:=Visu.ST00_245_S1_STOP,
					Reset:=gResetAll,
);

(* Call 	ST00_245_S2_START	Bedienstelle Produktion Start (DigIn) *)
ST00_245_S2_START(	sVisu:=Visu.ST00_245_S2_START,
					Reset:=gResetAll,
);

(* Call 	ST00_245_S3_RESET	Bedienstelle Produktion Reset (DigIn) *)
ST00_245_S3_RESET(	sVisu:=Visu.ST00_245_S3_RESET,
					Reset:=gResetAll,
);

(* ----------------------------------------------------------------------------------------- *)
(* 																				Ausgänge																					 *)
(* ----------------------------------------------------------------------------------------- *)

(* Call ST00_31_K1 Beleuchtung Anlage (DigOutIn) *)
ST00_31_K1(	sVisu:=Visu.ST00_31_K1,
			Reset:=gResetAll,
);

(* Call ST00_350_H1 Signalsäule RD Maschine Alarm/Störung (DigOutIn) *)
ST00_350_H1(sVisu:=Visu.ST00_350_H1,
			Reset:=gResetAll,
);

(* Call ST00_350_H2 Signalsäule YE Bedienereingriff erforderlich (DigOutIn) *)
ST00_350_H2(sVisu:=Visu.ST00_350_H2,
			Reset:=gResetAll,
);

(* Call ST00_350_H3 Signalsäule GN Maschine Automatik (DigOutIn) *) 
ST00_350_H3(sVisu:=Visu.ST00_350_H3,
			Reset:=gResetAll,
);

(* Call ST00_200_A1_E4 Quittierung Not-Aus (DigOutIn) *)
ST00_200_A1_E4(	sVisu:=Visu.ST00_200_A1_E4,
				Reset:=gResetAll,
);

(* Call ST00_220_S1_S31 Verriegelung Schutztüren (DigOutIn) *)
ST00_220_S1_S31                (sVisu:=Visu.ST00_220_S1_S31,
			Reset:=gResetAll,
);

(* Call ST00_292_H2_START Bedienstelle Start-Leuchte (DigOutIn) *)
ST00_292_H2_START(	sVisu:=Visu.ST00_292_H2_START,
					Reset:=gResetAll,
);

(* Call ST00_292_H3_RESET Bedienstelle Reset-Leuchte (DigOutIn) *)
ST00_292_H3_RESET(	sVisu:=Visu.ST00_292_H3_RESET,
					Reset:=gResetAll,
);

(* Call ST00_71_K2 Schnittstelle Bedrucken Tinte Abholposition frei (DigOutIn) *)
ST00_71_K2(	sVisu:=Visu.ST00_71_K2,
			Reset:=gResetAll,
);

(*  Call ST00_73_K3 Schnittstelle Förderband frei für Spritzmaschine*)
ST00_73_K3(	sVisu:=Visu.ST00_73_K3,
			Reset:=gResetAll,
);
(* Call ST00_73_K4   Schnittstelle Freigabe von Spritzmaschine (nur für Anlagen ohne Rundtisch) (DigIn) *)
ST00_73_K4(	sVisu:=Visu.ST00_73_K4,
			Reset:=gResetAll,
			CheckSignalHigh:=FALSE,
);
(* Call ST00_74_Y2_4 Vereinzeler Bandstrecke (Valve) *)
Analyze(	InputExp:=  TRUE,
			DoAnalyze:= TRUE );
ST00_74_Y2_4.strAnlayse:=Analyze.OutString;
ST00_74_Y2_4(	Enable  :=  Analyze.ExpResult,
				sVisu:=Visu.ST00_74_Y2_4,
				Reset:=gResetAll,
);
ST00_74_B7_2(ValveObject:= ADR(ST00_74_Y2_4));(*Vereinzeler GST1 DS*)
ST00_74_B7_3(ValveObject:= ADR(ST00_74_Y2_4));(*Vereinzeler GST2 PS*)


(* Call ST00_74_Y2_5 Vereinzeler Bandstrecke (Valve) *)
Analyze(	InputExp:=  TRUE,
			DoAnalyze:= TRUE );
ST00_74_Y2_5.strAnlayse:=Analyze.OutString;
ST00_74_Y2_5(	Enable  :=  Analyze.ExpResult,
				sVisu:=Visu.ST00_74_Y2_5,
				Reset:=gResetAll,
);
ST00_74_B7_4(ValveObject:= ADR(ST00_74_Y2_5));(*Vereinzeler AST1 DS*)
ST00_74_B7_6(ValveObject:= ADR(ST00_74_Y2_5));(*Vereinzeler GST1 DS*)
ST00_74_B7_5(ValveObject:= ADR(ST00_74_Y2_5));(*Vereinzeler AST2 PS*)
ST00_74_B7_7(ValveObject:= ADR(ST00_74_Y2_5));(*Vereinzeler GST2 PS*)
END_PROGRAM

(* POU Stations/ST_03_Ruestsaetze/ST_03_FBs/ST03_CallFBs, ST *)
PROGRAM ST03_CallFBs
VAR

	ST03_463_B70_3_4_pos	:INT;

END_VAR
(*Bei NOX4 darf der Override nicht größer 5 sein*)
IF gTypeCode=5631 AND MP.ST02.Override_Band>5 THEN
	MP.ST02.Override_Band:=5;
END_IF

(*Call ST03_51_M1 Förderbandmotor*)
ST03_51_M1			(sVisu:=Visu.ST03_51_M1,
						Override:= MP.ST02.Override_Band,
						Offset:=0,								(* in mm oder Grad am Abtrieb*)
						Reset:=gResetAll,
						NotausOK := TRUE);
(* ----------------------------------------------------------------------------------------- *)
(* 																	Roboter																									 *)
(* ----------------------------------------------------------------------------------------- *)

Robot01.sToolSettings.NameCoilA:='120_A1_A12';
Robot01.sToolSettings.NameCoilB:='xxxx';
Robot01.sToolSettings.NameInitSensor:='400_B12_4';
Robot01.sToolSettings.NameWorkSensor:='400_B12_5';
Robot01.sToolSettings.NameBtnToolOn:='Greifer Öffnen';
Robot01.sToolSettings.NameBtnToolOff:='Greifer Schliessen';

Analyze         (InputExp:=  ST03_Init_Lockings.InputExp_Robot01,
                 DoAnalyze:= TRUE );
Robot01(sVisu			:=visu.Robot01,
        Reset			:=gResetAll,
				Enable		:=TRUE,
				Acc				:=100,
				Vel				:=100,
				PosOffset :=gRobotOffset,
				strAnlayse:=Analyze.OutString,
				Override	:=MP.ST00.Override,
				CollisionActivated := MP.ST03.RoboterColisionActivated,
				Tool2Unit_AST :=ST03_400_B12_7.BitInToCheck);

(* ----------------------------------------------------------------------------------------- *)
(* 																	Eingänge																								 *)
(* ----------------------------------------------------------------------------------------- *)

(* Call ST03_125_F1 Absicherung Roboter iO (DigIn) *)
ST03_125_F1                    (sVisu:=Visu.ST03_125_F1,
                                Reset:=gResetAll,
																CheckSignalHigh:=TRUE,
);

(* Init ST03_A5 Bandantrieb Förderbandmotor Oriental (nur 3621) Ein (DigOutIn)*)
ST03_A5                  (sVisu:=Visu.ST03_A5,
                                Reset:=gResetAll,
);

(* Init ST03_601V1_A1 Förderband Prüfteile  (DigOutIn)*)
ST03_601V1_A1                  (sVisu:=Visu.ST03_601V1_A1,
                                Reset:=gResetAll,
);

(* Init ST03_V2 Störung Motor Förderband Oriental (DigIn) *)
ST03_V2                (sVisu:=Visu.ST03_V2,
                                Reset:=gResetAll,
);

(* Call ST03_120_A1:A14 Roboter Schwenkmodul ist ein (DigIn) *)
ST03_120_A1_A14                (sVisu:=Visu.ST03_120_A1_A14,
                                Reset:=gResetAll,
);

(* Call ST03_400_B12_6 Schwenkmodul AST (Roboterkopf) (DigIn) *)
ST03_400_B12_6                (sVisu:=Visu.ST03_400_B12_6,
                                Reset:=gResetAll,
);
(* Call ST03_400_B12_7 Schwenkmodul GST (Roboterkopf) (DigIn) *)
ST03_400_B12_7                (sVisu:=Visu.ST03_400_B12_7,
                                Reset:=gResetAll,
);
(* Call ST03_400_B54_7 Tray Testteile in Position (DigIn) *)
ST03_400_B54_7                (sVisu:=Visu.ST03_400_B54_7,
                                Reset:=gResetAll,
);
(* Call ST03_8_75_B13_5 voll/belegt keine Prüfmittel mehr (DigIn) *)
ST03_8_75_B13_5                (sVisu:=Visu.ST03_8_75_B13_5,
                                Reset:=gResetAll,
);
(* Call ST03_8_75_B13_6 belegt mit 6 Prüfmittel (DigIn) *)
ST03_8_75_B13_6                (sVisu:=Visu.ST03_8_75_B13_6,
                                Reset:=gResetAll,
);

(* Call ST03_BG3_X53_0 LED Taster Start Dummyprüfung Band (DigOutIn) *)
ST03_BG3_X53_0                  (sVisu:=Visu.ST03_BG3_X53_0,
                                Reset:=gResetAll,
);

(* Call ST03_65_Q1 Kühltunnel (Lüfter) (DigOutIn) *)
ST03_65_Q1                  (sVisu:=Visu.ST03_65_Q1,
                                Reset:=gResetAll,
);
(* Call ST03_65_F1 Sicherung Kühltunnel (Lüfter) *)
ST03_65_F1                (sVisu:=Visu.ST03_65_F1,
                                Reset:=gResetAll,
);

IF 	MP.ST03.SGM_3621 THEN
	(* Call ST03_Y01 Einschaltventil Hauptluft Tintenstrahldrucker (Valve) *)
	Analyze         (InputExp:=  TRUE,
	                 DoAnalyze:= TRUE );
	ST03_Y01.strAnlayse:=Analyze.OutString;
	ST03_Y01               (Enable  :=  Analyze.ExpResult,
	                                sVisu:=Visu.ST03_Y01,
	                                Reset:=gResetAll,
	);
END_IF

CASE  gTypeCode OF

4872:	call_154polRP();

4871:	call_154pol();

360, 379, 4992,489,322:	call_74_91_35_168_160pol();

522:		call_206pol();

550:		call_92pol();

564:		call_124pol();

569:		call_46pol();

5632,5633:	call_NOX5_6pol();

5631:	call_NOX4pol();

5731:	call_88pol();

575,5753,5754,5755:	call_7pol();

5732:	call_88polAMG();

5771:	call_120pol();

5772:	call_21pol();

580:	call_191pol();

5831:	call_72pol();

5832:	call_48pol();

5841, 4993:	call_268pol_102pol_neu();

5842:	call_268polRP();

598:	call_33pol();

END_CASE
END_PROGRAM
ACTION call_120pol:
(* Call ST03_531_B69_0 IZuführung  frei zum Ablegen ISK SP Maschine (DigIn) *)
ST03_531_B69_0(sVisu:=Visu.ST03_531_B69_0,
                                Reset:=gResetAll,
);
(* Call ST03_532_Y70_1  Zuführung Vereinzler AST/GST  (Valve) *)
Analyze(InputExp:=  TRUE, DoAnalyze:= TRUE );
ST03_532_Y70_1.strAnlayse:=Analyze.OutString;
ST03_532_Y70_1(Enable  :=  Analyze.ExpResult,
                                sVisu:=Visu.ST03_532_Y70_1,
                                Reset:=gResetAll,
);
ST03_531_B69_1(ValveObject:= ADR(ST03_532_Y70_1));(*  Zuführung Vereinzler eingefahren GST*)
ST03_531_B69_2(ValveObject:= ADR(ST03_532_Y70_1));(*  Zuführung Vereinzler ausgefahren AST*)

(* Call ST03_532_Y70_2  Züführung Stopper AST/GST  (Valve) *)
Analyze(InputExp:=  TRUE, DoAnalyze:= TRUE );
ST03_532_Y70_2.strAnlayse:=Analyze.OutString;
ST03_532_Y70_2(Enable  :=  Analyze.ExpResult,
                                sVisu:=Visu.ST03_532_Y70_2,
                                Reset:=gResetAll,
);
ST03_531_B69_3(ValveObject:= ADR(ST03_532_Y70_2));(* Zuführung Stopper  eingefahren  AST*)
ST03_531_B69_4(ValveObject:= ADR(ST03_532_Y70_2));(* Zuführung Stopper  ausgefahren GST*)


(* Call ST03_531_B69_6 SK anwesend am Stoper (DigIn) *)
ST03_531_B69_6(sVisu:=Visu.ST03_531_B69_6,
                                Reset:=gResetAll,
);
(* Call ST03_531_B69_7 ISK rechts Lageerkennung (DigIn) *)
ST03_531_B69_7(sVisu:=Visu.ST03_531_B69_7,
                                Reset:=gResetAll,
);
(* Call ST03_532_B70_0  ISK links Lageerkennung (DigIn) *)
ST03_532_B70_0(sVisu:=Visu.ST03_532_B70_0,
                                Reset:=gResetAll,
);
END_ACTION
ACTION call_124pol:
(* Call ST03_453_Y70_5 Förderband  Zuführung Vereinzler AST/GST  (Valve) *)
Analyze(InputExp:=  TRUE, DoAnalyze:= TRUE );
ST03_453_Y70_5.strAnlayse:=Analyze.OutString;
ST03_453_Y70_5(Enable  :=  Analyze.ExpResult,
                                sVisu:=Visu.ST03_453_Y70_5,
                                Reset:=gResetAll,
);
ST03_451_B69_0(ValveObject:= ADR(ST03_453_Y70_5));(*Förderband Zuführung Vereinzler   AST*)
ST03_451_B69_1(ValveObject:= ADR(ST03_453_Y70_5));(*Förderband Zuführung Vereinzler   GST*)

(* Call ST03_453_Y70_6 Förderband  Zuführung Stopper AST/GST  (Valve) *)
Analyze(InputExp:=  TRUE, DoAnalyze:= TRUE );
ST03_453_Y70_6.strAnlayse:=Analyze.OutString;
ST03_453_Y70_6(Enable  :=  Analyze.ExpResult,
                                sVisu:=Visu.ST03_453_Y70_6,
                                Reset:=gResetAll,
);
ST03_451_B69_2(ValveObject:= ADR(ST03_453_Y70_6));(*Förderband Zuführung Stopper   AST*)
ST03_451_B69_3(ValveObject:= ADR(ST03_453_Y70_6));(*Förderband Zuführung Stopper   GST*)

(* Call ST03_451_B69_4 Zuführung  frei zum Ablegen ISK SP Maschine Pos.1  (DigIn) *)
ST03_451_B69_4(sVisu:=Visu.ST03_451_B69_4,
                                Reset:=gResetAll,
);
(* Call ST03_451_B69_7 Zuführung  ISK anwesend am Stopper (DigIn) *)
ST03_451_B69_7(sVisu:=Visu.ST03_451_B69_7,
                                Reset:=gResetAll,
);
(* Call ST03_453_B70_4  ISK auf Übergabeposition zu Roboter  (DigIn) *)
ST03_453_B70_4(sVisu:=Visu.ST03_453_B70_4,
                                Reset:=gResetAll,
);
(* Call ST03_452_B70_1 Zuführung  ISK Lageerkennung links (DigIn) *)
ST03_452_B70_1(sVisu:=Visu.ST03_452_B70_1,
                                Reset:=gResetAll,
);
(* Call ST03_452_B70_2 Zuführung  ISK Lageerkennung links (DigIn) *)
ST03_452_B70_2(sVisu:=Visu.ST03_452_B70_2,
                                Reset:=gResetAll,
);
END_ACTION
ACTION call_154pol:
(* Call ST03_426_Y68_5 Förderband  Zuführung Vereinzler AST/GST  (Valve) *)
Analyze(InputExp:=  TRUE, DoAnalyze:= TRUE );
ST03_426_Y68_5.strAnlayse:=Analyze.OutString;
ST03_426_Y68_5(Enable  :=  Analyze.ExpResult,
                                sVisu:=Visu.ST03_426_Y68_5,
                                Reset:=gResetAll,
);
ST03_425_B67_0(ValveObject:= ADR(ST03_426_Y68_5));(*Förderband Zuführung Vereinzler   AST*)
ST03_425_B67_1(ValveObject:= ADR(ST03_426_Y68_5));(*Förderband Zuführung Vereinzler   GST*)

(* Call ST03_426_Y68_6 Förderband  Zuführung Stopper AST/GST  (Valve) *)
Analyze(InputExp:=  TRUE, DoAnalyze:= TRUE );
ST03_426_Y68_6.strAnlayse:=Analyze.OutString;
ST03_426_Y68_6(Enable  :=  Analyze.ExpResult,
                                sVisu:=Visu.ST03_426_Y68_6,
                                Reset:=gResetAll,
);
ST03_425_B67_2(ValveObject:= ADR(ST03_426_Y68_6));(*Förderband Zuführung Stopper   AST*)
ST03_425_B67_3(ValveObject:= ADR(ST03_426_Y68_6));(*Förderband Zuführung Stopper   GST*)

(* Call ST03_425_B67_4 Zuführung  frei zum Ablegen ISK SP Maschine Pos.1  (DigIn) *)
ST03_425_B67_4(sVisu:=Visu.ST03_425_B67_4,
                                Reset:=gResetAll,
);
(* Call ST03_425_B67_5 Zuführung  frei zum Ablegen ISK SP Maschine Pos.2  (DigIn) *)
ST03_425_B67_5(sVisu:=Visu.ST03_425_B67_5,
                                Reset:=gResetAll,
);
(* Call ST03_425_B67_6 Zuführung  frei zum Ablegen ISK SP Maschine Pos.3  (DigIn) *)
ST03_425_B67_6(sVisu:=Visu.ST03_425_B67_6,
                                Reset:=gResetAll,
);
(* Call ST03_425_B67_7 Zuführung  frei zum Ablegen ISK SP Maschine Pos.3  (DigIn) *)
ST03_425_B67_7(sVisu:=Visu.ST03_425_B67_7,
                                Reset:=gResetAll,
);
(* Call ST03_426_B68_4  ISK anwesend am Vereinzler  (DigIn) *)
ST03_426_B68_4(sVisu:=Visu.ST03_426_B68_4,
                                Reset:=gResetAll,
);
END_ACTION
ACTION call_154polRP:
(* Call ST03_418_B60_6 Zuführung links frei zum Ablegen ISK SP Maschine (DigIn) *)
ST03_418_B60_6(sVisu:=Visu.ST03_418_B60_6,
                                Reset:=gResetAll,
);
(* Call ST03_418_B60_7 Zuführung rechts frei zum Ablegen ISK SP Maschine (DigIn) *)
ST03_418_B60_7(sVisu:=Visu.ST03_418_B60_7,
                                Reset:=gResetAll,
);
(* Call ST03_419_B61_0 Förderband Zuführung links ISK anwesend zum Vereinzeln (DigIn) *)
ST03_419_B61_0(sVisu:=Visu.ST03_419_B61_0,
                                Reset:=gResetAll,
);
(* Call ST03_419_B61_1 Förderband Zuführung rechts ISK anwesend zum Vereinzeln (DigIn) *)
ST03_419_B61_1(sVisu:=Visu.ST03_419_B61_1,
                                Reset:=gResetAll,
);
(* Call ST03_419_B61_2 Züführung links ISK auf Übergabeposition Roboter Palettierer (DigIn) *)
ST03_419_B61_2(sVisu:=Visu.ST03_419_B61_2,
                                Reset:=gResetAll,
);
(* Call ST03_419_B61_3 Züführung rechts ISK auf Übergabeposition Roboter Palettierer (DigIn) *)
ST03_419_B61_3(sVisu:=Visu.ST03_419_B61_3,
                                Reset:=gResetAll,
);
(* Call ST03_419_Y61_5 Förderband linke Zuführung Vereinzler AST/GST  (Valve) *)
Analyze(InputExp:=  TRUE, DoAnalyze:= TRUE );
ST03_419_Y61_5.strAnlayse:=Analyze.OutString;
ST03_419_Y61_5(Enable  :=  Analyze.ExpResult,
                                sVisu:=Visu.ST03_419_Y61_5,
                                Reset:=gResetAll,
);
ST03_418_B60_0(ValveObject:= ADR(ST03_419_Y61_5));(*  Förderband linke Zuführung Vereinzler AST*)
ST03_418_B60_1(ValveObject:= ADR(ST03_419_Y61_5));(*  Förderband linke Zuführung Vereinzler GST*)

(* Call ST03_419_Y61_6 Förderband rechte Zuführung Vereinzler AST/GST  (Valve) *)
Analyze(InputExp:=  TRUE, DoAnalyze:= TRUE );
ST03_419_Y61_6.strAnlayse:=Analyze.OutString;
ST03_419_Y61_6(Enable  :=  Analyze.ExpResult,
                                sVisu:=Visu.ST03_419_Y61_6,
                                Reset:=gResetAll,
);
ST03_418_B60_2(ValveObject:= ADR(ST03_419_Y61_6));(*Förderband rechte Zuführung Vereinzler   AST*)
ST03_418_B60_3(ValveObject:= ADR(ST03_419_Y61_6));(*Förderband rechte Zuführung Vereinzler   GST*)

(* Call ST03_419_Y61_7 Förderband links/rechts Züführung Stopper AST/GST  (Valve) *)
Analyze(InputExp:=  TRUE, DoAnalyze:= TRUE );
ST03_419_Y61_7.strAnlayse:=Analyze.OutString;
ST03_419_Y61_7(Enable  :=  Analyze.ExpResult,
                                sVisu:=Visu.ST03_419_Y61_7,
                                Reset:=gResetAll,
);
ST03_418_B60_4(ValveObject:= ADR(ST03_419_Y61_7));(*Förderband links/rechts Zuführung Stopper   AST*)
ST03_418_B60_5(ValveObject:= ADR(ST03_419_Y61_7));(*Förderband links/rechts Zuführung Stopper   GST*)
END_ACTION
ACTION call_191pol:
(* Call ST03_541_B69_0 IZuführung  frei zum Ablegen ISK SP Maschine (DigIn) *)
ST03_541_B69_0(sVisu:=Visu.ST03_541_B69_0,
                                Reset:=gResetAll,
);
(* Call ST03_542_Y70_1  Zuführung Vereinzler AST/GST  (Valve) *)
Analyze(InputExp:=  TRUE, DoAnalyze:= TRUE );
ST03_542_Y70_1.strAnlayse:=Analyze.OutString;
ST03_542_Y70_1(Enable  :=  Analyze.ExpResult,
                                sVisu:=Visu.ST03_542_Y70_1,
                                Reset:=gResetAll,
);
ST03_541_B69_1(ValveObject:= ADR(ST03_542_Y70_1));(*  Zuführung Vereinzler eingefahren GST*)
ST03_541_B69_2(ValveObject:= ADR(ST03_542_Y70_1));(*  Zuführung Vereinzler ausgefahren AST*)

(* Call ST03_542_Y70_2  Züführung Stopper AST/GST  (Valve) *)
Analyze(InputExp:=  TRUE, DoAnalyze:= TRUE );
ST03_542_Y70_2.strAnlayse:=Analyze.OutString;
ST03_542_Y70_2(Enable  :=  Analyze.ExpResult,
                                sVisu:=Visu.ST03_542_Y70_2,
                                Reset:=gResetAll,
);
ST03_541_B69_3(ValveObject:= ADR(ST03_542_Y70_2));(* Zuführung Stopper  eingefahren  AST*)
ST03_541_B69_4(ValveObject:= ADR(ST03_542_Y70_2));(* Zuführung Stopper  ausgefahren GST*)


(* Call ST03_541_B69_6 SK anwesend am Stoper (DigIn) *)
ST03_541_B69_6(sVisu:=Visu.ST03_541_B69_6,
                                Reset:=gResetAll,
);
(* Call ST03_541_B69_7  ISK Lageerkennung links (DigIn) *)
ST03_541_B69_7(sVisu:=Visu.ST03_541_B69_7,
                                Reset:=gResetAll,
);
(* Call ST03_542_B70_0  ISK Lageerkennung rechts (DigIn) *)
ST03_542_B70_0(sVisu:=Visu.ST03_542_B70_0,
                                Reset:=gResetAll,
);
END_ACTION
ACTION call_206pol:
(* Call ST03_437_Y68_5 Förderband  Zuführung Vereinzler AST/GST  (Valve) *)
Analyze(InputExp:=  TRUE, DoAnalyze:= TRUE );
ST03_437_Y68_5.strAnlayse:=Analyze.OutString;
ST03_437_Y68_5(Enable  :=  Analyze.ExpResult,
                                sVisu:=Visu.ST03_437_Y68_5,
                                Reset:=gResetAll,
);
ST03_435_B67_0(ValveObject:= ADR(ST03_437_Y68_5));(*Förderband Zuführung Vereinzler   AST*)
ST03_435_B67_1(ValveObject:= ADR(ST03_437_Y68_5));(*Förderband Zuführung Vereinzler   GST*)

(* Call ST03_426_Y68_6 Förderband  Zuführung Stopper AST/GST  (Valve) *)
Analyze(InputExp:=  TRUE, DoAnalyze:= TRUE );
ST03_437_Y68_6.strAnlayse:=Analyze.OutString;
ST03_437_Y68_6(Enable  :=  Analyze.ExpResult,
                                sVisu:=Visu.ST03_437_Y68_6,
                                Reset:=gResetAll,
);
ST03_435_B67_2(ValveObject:= ADR(ST03_437_Y68_6));(*Förderband Zuführung Stopper   AST*)
ST03_435_B67_3(ValveObject:= ADR(ST03_437_Y68_6));(*Förderband Zuführung Stopper   GST*)

(* Call ST03_435_B67_4 Zuführung  frei zum Ablegen ISK SP Maschine Pos.1  (DigIn) *)
ST03_435_B67_4(sVisu:=Visu.ST03_435_B67_4,
                                Reset:=gResetAll,
);
(* Call ST03_435_B67_7 Zuführung  ISK anwesend am Stopper (DigIn) *)
ST03_435_B67_7(sVisu:=Visu.ST03_435_B67_7,
                                Reset:=gResetAll,
);
(* Call ST03_437_B68_4  ISK auf Übergabeposition zu Roboterr  (DigIn) *)
ST03_437_B68_4(sVisu:=Visu.ST03_437_B68_4,
                                Reset:=gResetAll,
);
(* Call ST03_436_B68_1 Zuführung  ISK Lageerkennung links (DigIn) *)
ST03_436_B68_1(sVisu:=Visu.ST03_436_B68_1,
                                Reset:=gResetAll,
);
(* Call ST03_436_B68_2 Zuführung  ISK Lageerkennung links (DigIn) *)
ST03_436_B68_2(sVisu:=Visu.ST03_436_B68_2,
                                Reset:=gResetAll,
);
END_ACTION
ACTION call_21pol:
(* Call ST03_536_B69_0 IZuführung  frei zum Ablegen ISK SP Maschine (DigIn) *)
ST03_536_B69_0(sVisu:=Visu.ST03_536_B69_0,
                                Reset:=gResetAll,
);
(* Call ST03_537_Y70_1  Zuführung Vereinzler AST/GST  (Valve) *)
Analyze(InputExp:=  TRUE, DoAnalyze:= TRUE );
ST03_537_Y70_1.strAnlayse:=Analyze.OutString;
ST03_537_Y70_1(Enable  :=  Analyze.ExpResult,
                                sVisu:=Visu.ST03_537_Y70_1,
                                Reset:=gResetAll,
);
ST03_536_B69_1(ValveObject:= ADR(ST03_537_Y70_1));(*  Zuführung Vereinzler eingefahren GST*)
ST03_536_B69_2(ValveObject:= ADR(ST03_537_Y70_1));(*  Zuführung Vereinzler ausgefahren AST*)

(* Call ST03_537_Y70_2  Züführung Stopper AST/GST  (Valve) *)
Analyze(InputExp:=  TRUE, DoAnalyze:= TRUE );
ST03_537_Y70_2.strAnlayse:=Analyze.OutString;
ST03_537_Y70_2(Enable  :=  Analyze.ExpResult,
                                sVisu:=Visu.ST03_537_Y70_2,
                                Reset:=gResetAll,
);
ST03_536_B69_3(ValveObject:= ADR(ST03_537_Y70_2));(* Zuführung Stopper  eingefahren  AST*)
ST03_536_B69_4(ValveObject:= ADR(ST03_537_Y70_2));(* Zuführung Stopper  ausgefahren GST*)


(* Call ST03_536_B69_6 SK anwesend am Stoper (DigIn) *)
ST03_536_B69_6(sVisu:=Visu.ST03_536_B69_6,
                                Reset:=gResetAll,
);
(* Call ST03_536_B69_7 ISK anwesend an Abholposition (DigIn) *)
ST03_536_B69_7(sVisu:=Visu.ST03_536_B69_7,
                                Reset:=gResetAll,
);
(* Call ST03_537_B70_0  ISK Lageerkennung (DigIn) *)
ST03_537_B70_0(sVisu:=Visu.ST03_537_B70_0,
                                Reset:=gResetAll,
);
END_ACTION
ACTION call_268pol_102pol_neu:
ST03_8_100_A1(
		Activated := MP.ST03.CamOn[1],
		st_InstName:='ST03_8_100_A1',
		st_Description:= 'Kamera 1 Farberkennung',
		SensopartErgebnis:=TD.SensopartErgebnis,
		);
ST03_8_100_A1.s_IpAdress := MP.ST03.SensopartIPAdress[1];  		(* 'MP.SensopartIPAdress';*)
ST03_8_100_A1.i_CmdPort := 2006;
ST03_8_100_A1.i_DataPort :=2005;

IF	gTypeCode = 4993 THEN
	ST03_8_103_A1(
			Activated := MP.ST03.CamOn[2],
			st_InstName:='ST03_8_103_A1',
			st_Description:= 'Kamera 2 Flügelerkennung',
			SensopartErgebnis:=TD.Sensopart2Ergebnis,
			);
	ST03_8_103_A1.s_IpAdress := MP.ST03.SensopartIPAdress[2];  		(* 'MP.SensopartIPAdress';*)
	ST03_8_103_A1.i_CmdPort := 2006;
	ST03_8_103_A1.i_DataPort :=2005;
END_IF


(* Call ST03_556_B69_0 IZuführung  frei zum Ablegen ISK SP Maschine (DigIn) *)
ST03_556_B69_0(sVisu:=Visu.ST03_556_B69_0,
                                Reset:=gResetAll,
);
(* Call ST03_556_Y70_1  Zuführung Vereinzler AST/GST  (Valve) *)
Analyze(InputExp:=  TRUE, DoAnalyze:= TRUE );
ST03_557_Y70_1.strAnlayse:=Analyze.OutString;
ST03_557_Y70_1(Enable  :=  Analyze.ExpResult,
                                sVisu:=Visu.ST03_557_Y70_1,
                                Reset:=gResetAll,
);
ST03_556_B69_1(ValveObject:= ADR(ST03_557_Y70_1));(*  Zuführung Vereinzler eingefahren GST*)
ST03_556_B69_2(ValveObject:= ADR(ST03_557_Y70_1));(*  Zuführung Vereinzler ausgefahren AST*)

(* Call ST03_556_Y70_2  Züführung Stopper AST/GST  (Valve) *)
Analyze(InputExp:=  TRUE, DoAnalyze:= TRUE );
ST03_557_Y70_2.strAnlayse:=Analyze.OutString;
ST03_557_Y70_2(Enable  :=  Analyze.ExpResult,
                                sVisu:=Visu.ST03_557_Y70_2,
                                Reset:=gResetAll,
);
ST03_556_B69_3(ValveObject:= ADR(ST03_557_Y70_2));(* Zuführung Stopper  eingefahren  AST*)
ST03_556_B69_4(ValveObject:= ADR(ST03_557_Y70_2));(* Zuführung Stopper  ausgefahren GST*)

(* Call ST03_556_B69_5 Führungsschiene Überwachung Staustrecke (DigIn) *)
ST03_556_B69_5(sVisu:=Visu.ST03_556_B69_5,
                                Reset:=gResetAll,
);

(* Call ST03_556_B69_6 SK anwesend am Stoper (DigIn) *)
ST03_556_B69_6(sVisu:=Visu.ST03_556_B69_6,
                                Reset:=gResetAll,
);
(* Call ST03_546_B69_7 ISK  auf Übergabeposition  (DigIn) *)
ST03_556_B69_7(sVisu:=Visu.ST03_556_B69_7,
                                Reset:=gResetAll,
);
END_ACTION
ACTION call_268polRP:
(*Rüstsatz 268 pol Rasterplatte======================================================================================*)

(* Call ST03_562_B69_0 Zuführung 1 frei zum schwenken (DigIn) *)
ST03_562_B69_0(sVisu:=Visu.ST03_562_B69_0,
                                Reset:=gResetAll,
);
(* Call ST03_562_B69_6 Zuführung 1 ISK anwesend am Stopper (DigIn) *)
ST03_562_B69_6(sVisu:=Visu.ST03_562_B69_6,
                                Reset:=gResetAll,
);
(* Call ST03_562_B67_7 Zuführung 1 ISK auf Übergabepos. Robi (DigIn) *)
ST03_562_B67_7(sVisu:=Visu.ST03_562_B67_7,
                                Reset:=gResetAll,
);
(* Call ST03_563_B70_0 Zuführung 2 frei zum schwenken (DigIn) *)
ST03_563_B70_0(sVisu:=Visu.ST03_563_B70_0,
                                Reset:=gResetAll,
);
(* Call ST03_563_B70_6 Zuführung 2 ISK anwesend am Stopper (DigIn) *)
ST03_563_B70_6(sVisu:=Visu.ST03_563_B70_6,
                                Reset:=gResetAll,
);
(* Call ST03_563_B70_7 Zuführung 2 ISK auf Übergabepos. Robi (DigIn) *)
ST03_563_B70_7(sVisu:=Visu.ST03_563_B70_7,
                                Reset:=gResetAll,
);
(* Call ST03_565_B72_0 ISK 1 in Klemmer (DigIn) *)
ST03_565_B72_0(sVisu:=Visu.ST03_565_B72_0,
                                Reset:=gResetAll,
);
(* Call ST03_565_B72_1 ISK 2 in Klemmer (DigIn) *)
ST03_565_B72_1(sVisu:=Visu.ST03_565_B72_1,
                                Reset:=gResetAll,
);
(* Call ST03_564_Y71_0 Zuführung 1 Vereinzler AST/GST  (Valve) *)
Analyze(InputExp:=  TRUE, DoAnalyze:= TRUE );
ST03_564_Y71_0.strAnlayse:=Analyze.OutString;
ST03_564_Y71_0(Enable  :=  Analyze.ExpResult,
                                sVisu:=Visu.ST03_564_Y71_0,
                                Reset:=gResetAll,
);
ST03_562_B69_1(ValveObject:= ADR(ST03_564_Y71_0));(*Zuführung 1 Zuführung Vereinzler AST*)
ST03_562_B69_2(ValveObject:= ADR(ST03_564_Y71_0));(*Zuführung 1 Zuführung Vereinzler GST*)

(* Call ST03_564_Y71_1 Zuführung 1 Stopper AST/GST  (Valve) *)
Analyze(InputExp:=  TRUE, DoAnalyze:= TRUE );
ST03_564_Y71_1.strAnlayse:=Analyze.OutString;
ST03_564_Y71_1(Enable  :=  Analyze.ExpResult,
                                sVisu:=Visu.ST03_564_Y71_1,
                                Reset:=gResetAll,
);
ST03_562_B69_3(ValveObject:= ADR(ST03_564_Y71_1));(*Zuführung 1 Zuführung Stopper AST*)
ST03_562_B69_4(ValveObject:= ADR(ST03_564_Y71_1));(*Zuführung 1 Zuführung Stopper GST*)

(* Call ST03_564_Y71_2 Zuführung 2 Vereinzler AST/GST  (Valve) *)
Analyze(InputExp:=  TRUE, DoAnalyze:= TRUE );
ST03_564_Y71_2.strAnlayse:=Analyze.OutString;
ST03_564_Y71_2(Enable  :=  Analyze.ExpResult,
                                sVisu:=Visu.ST03_564_Y71_2,
                                Reset:=gResetAll,
);
ST03_563_B70_1(ValveObject:= ADR(ST03_564_Y71_2));(*Zuführung 2 Zuführung Vereinzler AST*)
ST03_563_B70_2(ValveObject:= ADR(ST03_564_Y71_2));(*Zuführung 2 Zuführung Vereinzler GST*)

(* Call ST03_564_Y71_3 Zuführung 2 Stopper AST/GST  (Valve) *)
Analyze(InputExp:=  TRUE, DoAnalyze:= TRUE );
ST03_564_Y71_3.strAnlayse:=Analyze.OutString;
ST03_564_Y71_3(Enable  :=  Analyze.ExpResult,
                                sVisu:=Visu.ST03_564_Y71_3,
                                Reset:=gResetAll,
);
ST03_563_B70_3(ValveObject:= ADR(ST03_564_Y71_3));(*Zuführung 2 Zuführung Stopper AST*)
ST03_563_B70_4(ValveObject:= ADR(ST03_564_Y71_3));(*Zuführung 2 Zuführung Stopper GST*)


(* Call ST03_564_Y71_4 ISK Klemmer  AST/GST  (Valve) *)
Analyze(InputExp:=  TRUE, DoAnalyze:= TRUE );
ST03_564_Y71_4.strAnlayse:=Analyze.OutString;
ST03_564_Y71_4(Enable  :=  Analyze.ExpResult,
                                sVisu:=Visu.ST03_564_Y71_4,
                                Reset:=gResetAll,
);
ST03_565_B72_4(ValveObject:= ADR(ST03_564_Y71_4));(*ISK Klemmer 2 offen GST*)
ST03_565_B72_5(ValveObject:= ADR(ST03_564_Y71_4));(*ISK Klemmer 2 zu AST*)
ST03_565_B72_2(ValveObject:= ADR(ST03_564_Y71_4));(*ISK Klemmer 1 offen GST*)
ST03_565_B72_3(ValveObject:= ADR(ST03_564_Y71_4));(*ISK Klemmer 1 zu AST*)

(* Call ST03_564_Y71_5 Rinne schwenkern AST/GST  (Valve) *)
Analyze(InputExp:=  TRUE, DoAnalyze:= TRUE );
ST03_564_Y71_5.strAnlayse:=Analyze.OutString;
ST03_564_Y71_5(Enable  :=  Analyze.ExpResult,
                                sVisu:=Visu.ST03_564_Y71_5,
                                Reset:=gResetAll,
);
ST03_565_B72_6(ValveObject:= ADR(ST03_564_Y71_5));(*ISK Klemmer schwenkern 0° AST*)
ST03_565_B72_7(ValveObject:= ADR(ST03_564_Y71_5));(*ISK Klemmer schwenkern 180° GST*)
END_ACTION
ACTION call_33pol:
(* Call ST03_571_B69_0 Zuführung Pos 1  frei zum Ablegen ISK SP Maschine (DigIn) *)
ST03_571_B69_0(sVisu:=Visu.ST03_571_B69_0,
                                Reset:=gResetAll,
);
(* Call ST03_571_B69_1 Zuführung Pos 2  frei zum Ablegen ISK SP Maschine (DigIn) *)
ST03_571_B69_1(sVisu:=Visu.ST03_571_B69_1,
                                Reset:=gResetAll,
);

